LIN {X 42.103,Y -31.707,Z -45.890,A -90.000,B 90.000,C 0.000} C_DIS
LIN {X 42.764,Y -31.745,Z -45.727,A -90.000,B 90.000,C 0.000} C_DIS
LIN {X 43.314,Y -31.756,Z -45.575,A -90.000,B 90.000,C 0.000} C_DIS
LIN {X 43.681,Y -31.756,Z -45.477,A -90.000,B 90.000,C 0.000} C_DIS
LIN {X 44.130,Y -31.751,Z -45.363,A -90.000,B 90.000,C 0.000} C_DIS
LIN {X 44.222,Y -31.752,Z -45.341,A -90.000,B 90.000,C 0.000} C_DIS
LIN {X 44.913,Y -31.771,Z -45.188,A -90.000,B 90.000,C 0.000} C_DIS
LIN {X 45.364,Y -31.765,Z -45.111,A -90.000,B 90.000,C 0.000} C_DIS
LIN {X 45.432,Y -31.762,Z -45.099,A -90.000,B 90.000,C 0.000} C_DIS
LIN {X 45.844,Y -31.730,Z -45.045,A -90.000,B 90.000,C 0.000} C_DIS
LIN {X 45.937,Y -31.721,Z -45.037,A -90.000,B 90.000,C 0.000} C_DIS
LIN {X 46.177,Y -31.703,Z -45.019,A -90.000,B 90.000,C 0.000} C_DIS
LIN {X 46.589,Y -31.686,Z -44.979,A -90.000,B 90.000,C 0.000} C_DIS
LIN {X 46.721,Y -31.684,Z -44.970,A -90.000,B 90.000,C 0.000} C_DIS
LIN {X 47.117,Y -31.682,Z -44.943,A -90.000,B 90.000,C 0.000} C_DIS
LIN {X 47.760,Y -31.692,Z -44.913,A -90.000,B 90.000,C 0.000} C_DIS
LIN {X 48.195,Y -31.687,Z -44.927,A -90.000,B 90.000,C 0.000} C_DIS
LIN {X 48.804,Y -31.665,Z -44.973,A -90.000,B 90.000,C 0.000} C_DIS
LIN {X 49.258,Y -31.648,Z -45.032,A -90.000,B 90.000,C 0.000} C_DIS
LIN {X 49.697,Y -31.626,Z -45.108,A -90.000,B 90.000,C 0.000} C_DIS
LIN {X 49.817,Y -31.620,Z -45.134,A -90.000,B 90.000,C 0.000} C_DIS
LIN {X 50.403,Y -31.602,Z -45.264,A -90.000,B 90.000,C 0.000} C_DIS
LIN {X 50.513,Y -31.602,Z -45.290,A -90.000,B 90.000,C 0.000} C_DIS
LIN {X 50.923,Y -31.594,Z -45.415,A -90.000,B 90.000,C 0.000} C_DIS
LIN {X 51.695,Y -31.586,Z -45.677,A -90.000,B 90.000,C 0.000} C_DIS
LIN {X 52.507,Y -31.561,Z -46.005,A -90.000,B 90.000,C 0.000} C_DIS
LIN {X 52.949,Y -31.557,Z -46.198,A -90.000,B 90.000,C 0.000} C_DIS
LIN {X 53.402,Y -31.550,Z -46.401,A -90.000,B 90.000,C 0.000} C_DIS
LIN {X 53.812,Y -31.543,Z -46.594,A -90.000,B 90.000,C 0.000} C_DIS
LIN {X 54.024,Y -31.537,Z -46.700,A -90.000,B 90.000,C 0.000} C_DIS
LIN {X 54.190,Y -31.540,Z -46.786,A -90.000,B 90.000,C 0.000} C_DIS
LIN {X 54.466,Y -31.543,Z -46.938,A -90.000,B 90.000,C 0.000} C_DIS
LIN {X 54.513,Y -31.543,Z -46.967,A -90.000,B 90.000,C 0.000} C_DIS
LIN {X 54.861,Y -31.548,Z -47.185,A -90.000,B 90.000,C 0.000} C_DIS
LIN {X 55.840,Y -31.525,Z -47.889,A -90.000,B 90.000,C 0.000} C_DIS
LIN {X 57.235,Y -31.497,Z -48.888,A -90.000,B 90.000,C 0.000} C_DIS
LIN {X 57.411,Y -31.498,Z -49.016,A -90.000,B 90.000,C 0.000} C_DIS
LIN {X 57.592,Y -31.496,Z -49.156,A -90.000,B 90.000,C 0.000} C_DIS
LIN {X 57.780,Y -31.499,Z -49.303,A -90.000,B 90.000,C 0.000} C_DIS
LIN {X 59.169,Y -31.488,Z -50.515,A -90.000,B 90.000,C 0.000} C_DIS
LIN {X 60.060,Y -31.484,Z -51.286,A -90.000,B 90.000,C 0.000} C_DIS
LIN {X 60.371,Y -31.483,Z -51.578,A -90.000,B 90.000,C 0.000} C_DIS
LIN {X 61.487,Y -31.484,Z -52.631,A -90.000,B 90.000,C 0.000} C_DIS
LIN {X 62.016,Y -31.485,Z -53.126,A -90.000,B 90.000,C 0.000} C_DIS
LIN {X 62.615,Y -31.489,Z -53.684,A -90.000,B 90.000,C 0.000} C_DIS
LIN {X 63.420,Y -31.498,Z -54.433,A -90.000,B 90.000,C 0.000} C_DIS
LIN {X 64.379,Y -31.509,Z -55.331,A -90.000,B 90.000,C 0.000} C_DIS
LIN {X 64.718,Y -31.523,Z -55.625,A -90.000,B 90.000,C 0.000} C_DIS
LIN {X 65.056,Y -31.534,Z -55.917,A -90.000,B 90.000,C 0.000} C_DIS
LIN {X 65.997,Y -31.557,Z -56.726,A -90.000,B 90.000,C 0.000} C_DIS
LIN {X 66.900,Y -31.586,Z -57.486,A -90.000,B 90.000,C 0.000} C_DIS
LIN {X 67.393,Y -31.606,Z -57.902,A -90.000,B 90.000,C 0.000} C_DIS
LIN {X 68.612,Y -31.651,Z -58.950,A -90.000,B 90.000,C 0.000} C_DIS
LIN {X 69.045,Y -31.655,Z -59.347,A -90.000,B 90.000,C 0.000} C_DIS
LIN {X 69.869,Y -31.693,Z -60.129,A -90.000,B 90.000,C 0.000} C_DIS
LIN {X 70.229,Y -31.703,Z -60.488,A -90.000,B 90.000,C 0.000} C_DIS
LIN {X 70.602,Y -31.727,Z -60.873,A -90.000,B 90.000,C 0.000} C_DIS
LIN {X 71.184,Y -31.746,Z -61.521,A -90.000,B 90.000,C 0.000} C_DIS
LIN {X 72.241,Y -31.804,Z -62.721,A -90.000,B 90.000,C 0.000} C_DIS
LIN {X 72.515,Y -31.817,Z -63.037,A -90.000,B 90.000,C 0.000} C_DIS
LIN {X 72.609,Y -31.817,Z -63.151,A -90.000,B 90.000,C 0.000} C_DIS
LIN {X 72.801,Y -31.813,Z -63.398,A -90.000,B 90.000,C 0.000} C_DIS
LIN {X 72.929,Y -31.812,Z -63.565,A -90.000,B 90.000,C 0.000} C_DIS
LIN {X 73.104,Y -31.812,Z -63.793,A -90.000,B 90.000,C 0.000} C_DIS
LIN {X 73.529,Y -31.818,Z -64.361,A -90.000,B 90.000,C 0.000} C_DIS
LIN {X 73.683,Y -31.819,Z -64.579,A -90.000,B 90.000,C 0.000} C_DIS
LIN {X 73.927,Y -31.829,Z -64.916,A -90.000,B 90.000,C 0.000} C_DIS
LIN {X 73.994,Y -31.828,Z -65.015,A -90.000,B 90.000,C 0.000} C_DIS
LIN {X 74.219,Y -31.808,Z -65.329,A -90.000,B 90.000,C 0.000} C_DIS
LIN {X 74.431,Y -31.799,Z -65.639,A -90.000,B 90.000,C 0.000} C_DIS
LIN {X 74.577,Y -31.806,Z -65.839,A -90.000,B 90.000,C 0.000} C_DIS
LIN {X 74.823,Y -31.798,Z -66.153,A -90.000,B 90.000,C 0.000} C_DIS
LIN {X 74.927,Y -31.796,Z -66.289,A -90.000,B 90.000,C 0.000} C_DIS
LIN {X 75.187,Y -31.788,Z -66.638,A -90.000,B 90.000,C 0.000} C_DIS
LIN {X 75.305,Y -31.780,Z -66.797,A -90.000,B 90.000,C 0.000} C_DIS
LIN {X 75.814,Y -31.762,Z -67.510,A -90.000,B 90.000,C 0.000} C_DIS
LIN {X 75.836,Y -31.763,Z -67.538,A -90.000,B 90.000,C 0.000} C_DIS
LIN {X 75.961,Y -31.757,Z -67.682,A -90.000,B 90.000,C 0.000} C_DIS
LIN {X 76.227,Y -31.729,Z -68.017,A -90.000,B 90.000,C 0.000} C_DIS
LIN {X 76.293,Y -31.724,Z -68.107,A -90.000,B 90.000,C 0.000} C_DIS
LIN {X 76.429,Y -31.718,Z -68.299,A -90.000,B 90.000,C 0.000} C_DIS
LIN {X 76.455,Y -31.719,Z -68.332,A -90.000,B 90.000,C 0.000} C_DIS
LIN {X 76.904,Y -31.702,Z -68.861,A -90.000,B 90.000,C 0.000} C_DIS
LIN {X 76.997,Y -31.696,Z -68.977,A -90.000,B 90.000,C 0.000} C_DIS
LIN {X 77.105,Y -31.691,Z -69.109,A -90.000,B 90.000,C 0.000} C_DIS
LIN {X 77.203,Y -31.686,Z -69.228,A -90.000,B 90.000,C 0.000} C_DIS
LIN {X 77.430,Y -31.682,Z -69.512,A -90.000,B 90.000,C 0.000} C_DIS
LIN {X 77.622,Y -31.678,Z -69.759,A -90.000,B 90.000,C 0.000} C_DIS
LIN {X 77.717,Y -31.609,Z -69.804,A -90.000,B 90.000,C 0.000} C_DIS
LIN {X 77.780,Y -31.567,Z -69.838,A -90.000,B 90.000,C 0.000} C_DIS
LIN {X 77.852,Y -31.523,Z -69.884,A -90.000,B 90.000,C 0.000} C_DIS
LIN {X 77.939,Y -31.475,Z -69.946,A -90.000,B 90.000,C 0.000} C_DIS
LIN {X 78.032,Y -31.430,Z -70.019,A -90.000,B 90.000,C 0.000} C_DIS
LIN {X 78.096,Y -31.404,Z -70.072,A -90.000,B 90.000,C 0.000} C_DIS
LIN {X 78.244,Y -31.354,Z -70.211,A -90.000,B 90.000,C 0.000} C_DIS
LIN {X 78.265,Y -31.349,Z -70.232,A -90.000,B 90.000,C 0.000} C_DIS
LIN {X 78.399,Y -31.321,Z -70.376,A -90.000,B 90.000,C 0.000} C_DIS
LIN {X 78.478,Y -31.312,Z -70.466,A -90.000,B 90.000,C 0.000} C_DIS
LIN {X 78.570,Y -31.308,Z -70.580,A -90.000,B 90.000,C 0.000} C_DIS
LIN {X 78.560,Y -31.341,Z -70.590,A -90.000,B 90.000,C 0.000} C_DIS
LIN {X 78.561,Y -35.835,Z -70.592,A -90.000,B 90.000,C 0.000} C_DIS
LIN {X 78.567,Y -36.729,Z -70.599,A -90.000,B 90.000,C 0.000} C_DIS
LIN {X 78.574,Y -37.040,Z -70.607,A -90.000,B 90.000,C 0.000} C_DIS
LIN {X 78.584,Y -37.233,Z -70.617,A -90.000,B 90.000,C 0.000} C_DIS
LIN {X 78.578,Y -37.064,Z -70.596,A -90.000,B 90.000,C 0.000} C_DIS
LIN {X 78.575,Y -36.863,Z -70.579,A -90.000,B 90.000,C 0.000} C_DIS
LIN {X 78.573,Y -35.838,Z -70.554,A -90.000,B 90.000,C 0.000} C_DIS
LIN {X 78.573,Y -31.307,Z -70.553,A -90.000,B 90.000,C 0.000} C_DIS
LIN {X 78.577,Y -31.307,Z -70.516,A -90.000,B 90.000,C 0.000} C_DIS
LIN {X 78.594,Y -31.308,Z -70.505,A -90.000,B 90.000,C 0.000} C_DIS
LIN {X 78.624,Y -31.308,Z -70.415,A -90.000,B 90.000,C 0.000} C_DIS
LIN {X 78.683,Y -36.449,Z -70.235,A -90.000,B 90.000,C 0.000} C_DIS
LIN {X 78.690,Y -36.457,Z -70.213,A -90.000,B 90.000,C 0.000} C_DIS
LIN {X 78.691,Y -36.460,Z -70.211,A -90.000,B 90.000,C 0.000} C_DIS
LIN {X 78.693,Y -36.503,Z -70.206,A -90.000,B 90.000,C 0.000} C_DIS
LIN {X 78.701,Y -36.545,Z -70.184,A -90.000,B 90.000,C 0.000} C_DIS
LIN {X 78.761,Y -31.308,Z -70.004,A -90.000,B 90.000,C 0.000} C_DIS
LIN {X 78.774,Y -31.308,Z -69.967,A -90.000,B 90.000,C 0.000} C_DIS
LIN {X 78.774,Y -60.000,Z -69.967,A -90.000,B 90.000,C 0.000} C_DIS
LIN {X 87.886,Y -60.000,Z -55.601,A -90.000,B 90.000,C 0.000} C_DIS
LIN {X 87.886,Y -31.308,Z -55.601,A -90.000,B 90.000,C 0.000} C_DIS
LIN {X 87.895,Y -31.310,Z -55.489,A -90.000,B 90.000,C 0.000} C_DIS
LIN {X 87.955,Y -31.321,Z -55.235,A -90.000,B 90.000,C 0.000} C_DIS
LIN {X 88.019,Y -31.333,Z -55.056,A -90.000,B 90.000,C 0.000} C_DIS
LIN {X 88.137,Y -31.354,Z -54.797,A -90.000,B 90.000,C 0.000} C_DIS
LIN {X 88.416,Y -31.405,Z -54.284,A -90.000,B 90.000,C 0.000} C_DIS
LIN {X 88.556,Y -31.441,Z -54.017,A -90.000,B 90.000,C 0.000} C_DIS
LIN {X 88.594,Y -31.451,Z -53.947,A -90.000,B 90.000,C 0.000} C_DIS
LIN {X 88.969,Y -31.547,Z -53.327,A -90.000,B 90.000,C 0.000} C_DIS
LIN {X 89.043,Y -31.566,Z -53.212,A -90.000,B 90.000,C 0.000} C_DIS
LIN {X 89.236,Y -31.615,Z -52.925,A -90.000,B 90.000,C 0.000} C_DIS
LIN {X 89.391,Y -31.655,Z -52.704,A -90.000,B 90.000,C 0.000} C_DIS
LIN {X 89.464,Y -31.674,Z -52.605,A -90.000,B 90.000,C 0.000} C_DIS
LIN {X 89.839,Y -31.793,Z -52.083,A -90.000,B 90.000,C 0.000} C_DIS
LIN {X 90.193,Y -31.904,Z -51.622,A -90.000,B 90.000,C 0.000} C_DIS
LIN {X 90.500,Y -32.000,Z -51.242,A -90.000,B 90.000,C 0.000} C_DIS
LIN {X 90.638,Y -32.043,Z -51.076,A -90.000,B 90.000,C 0.000} C_DIS
LIN {X 91.176,Y -32.230,Z -50.436,A -90.000,B 90.000,C 0.000} C_DIS
LIN {X 91.462,Y -32.330,Z -50.116,A -90.000,B 90.000,C 0.000} C_DIS
LIN {X 91.851,Y -32.466,Z -49.697,A -90.000,B 90.000,C 0.000} C_DIS
LIN {X 92.169,Y -32.589,Z -49.359,A -90.000,B 90.000,C 0.000} C_DIS
LIN {X 92.399,Y -32.678,Z -49.123,A -90.000,B 90.000,C 0.000} C_DIS
LIN {X 92.339,Y -32.668,Z -48.928,A -90.000,B 90.000,C 0.000} C_DIS
LIN {X 92.298,Y -32.662,Z -48.770,A -90.000,B 90.000,C 0.000} C_DIS
LIN {X 92.252,Y -32.641,Z -48.535,A -90.000,B 90.000,C 0.000} C_DIS
LIN {X 92.218,Y -32.617,Z -48.349,A -90.000,B 90.000,C 0.000} C_DIS
LIN {X 92.177,Y -32.587,Z -48.082,A -90.000,B 90.000,C 0.000} C_DIS
LIN {X 92.166,Y -32.569,Z -47.976,A -90.000,B 90.000,C 0.000} C_DIS
LIN {X 92.158,Y -32.552,Z -47.869,A -90.000,B 90.000,C 0.000} C_DIS
LIN {X 92.148,Y -32.512,Z -47.664,A -90.000,B 90.000,C 0.000} C_DIS
LIN {X 92.146,Y -32.500,Z -47.597,A -90.000,B 90.000,C 0.000} C_DIS
LIN {X 92.150,Y -32.478,Z -47.451,A -90.000,B 90.000,C 0.000} C_DIS
LIN {X 92.171,Y -32.438,Z -47.211,A -90.000,B 90.000,C 0.000} C_DIS
LIN {X 92.200,Y -32.388,Z -46.981,A -90.000,B 90.000,C 0.000} C_DIS
LIN {X 92.221,Y -32.361,Z -46.845,A -90.000,B 90.000,C 0.000} C_DIS
LIN {X 92.284,Y -32.302,Z -46.521,A -90.000,B 90.000,C 0.000} C_DIS
LIN {X 92.307,Y -32.284,Z -46.424,A -90.000,B 90.000,C 0.000} C_DIS
LIN {X 92.324,Y -32.273,Z -46.362,A -90.000,B 90.000,C 0.000} C_DIS
LIN {X 92.409,Y -32.240,Z -46.102,A -90.000,B 90.000,C 0.000} C_DIS
LIN {X 92.452,Y -32.221,Z -45.979,A -90.000,B 90.000,C 0.000} C_DIS
LIN {X 92.675,Y -32.135,Z -45.409,A -90.000,B 90.000,C 0.000} C_DIS
LIN {X 92.727,Y -32.118,Z -45.300,A -90.000,B 90.000,C 0.000} C_DIS
LIN {X 92.805,Y -32.095,Z -45.145,A -90.000,B 90.000,C 0.000} C_DIS
LIN {X 92.914,Y -32.062,Z -44.937,A -90.000,B 90.000,C 0.000} C_DIS
LIN {X 93.148,Y -32.006,Z -44.518,A -90.000,B 90.000,C 0.000} C_DIS
LIN {X 93.166,Y -32.002,Z -44.486,A -90.000,B 90.000,C 0.000} C_DIS
LIN {X 93.389,Y -31.943,Z -44.141,A -90.000,B 90.000,C 0.000} C_DIS
LIN {X 93.591,Y -31.898,Z -43.848,A -90.000,B 90.000,C 0.000} C_DIS
LIN {X 93.761,Y -31.866,Z -43.610,A -90.000,B 90.000,C 0.000} C_DIS
LIN {X 94.205,Y -31.773,Z -43.062,A -90.000,B 90.000,C 0.000} C_DIS
LIN {X 94.307,Y -31.752,Z -42.942,A -90.000,B 90.000,C 0.000} C_DIS
LIN {X 94.451,Y -31.729,Z -42.780,A -90.000,B 90.000,C 0.000} C_DIS
LIN {X 94.667,Y -31.693,Z -42.552,A -90.000,B 90.000,C 0.000} C_DIS
LIN {X 94.923,Y -31.657,Z -42.285,A -90.000,B 90.000,C 0.000} C_DIS
LIN {X 95.182,Y -31.617,Z -42.030,A -90.000,B 90.000,C 0.000} C_DIS
LIN {X 95.304,Y -31.603,Z -41.920,A -90.000,B 90.000,C 0.000} C_DIS
LIN {X 95.776,Y -31.549,Z -41.516,A -90.000,B 90.000,C 0.000} C_DIS
LIN {X 95.980,Y -31.527,Z -41.343,A -90.000,B 90.000,C 0.000} C_DIS
LIN {X 96.207,Y -31.500,Z -41.168,A -90.000,B 90.000,C 0.000} C_DIS
LIN {X 96.826,Y -31.455,Z -40.703,A -90.000,B 90.000,C 0.000} C_DIS
LIN {X 96.924,Y -31.447,Z -40.637,A -90.000,B 90.000,C 0.000} C_DIS
LIN {X 97.187,Y -31.423,Z -40.470,A -90.000,B 90.000,C 0.000} C_DIS
LIN {X 97.655,Y -31.396,Z -40.178,A -90.000,B 90.000,C 0.000} C_DIS
LIN {X 98.035,Y -31.375,Z -39.949,A -90.000,B 90.000,C 0.000} C_DIS
LIN {X 98.217,Y -31.365,Z -39.850,A -90.000,B 90.000,C 0.000} C_DIS
LIN {X 98.843,Y -31.345,Z -39.508,A -90.000,B 90.000,C 0.000} C_DIS
LIN {X 99.070,Y -31.336,Z -39.398,A -90.000,B 90.000,C 0.000} C_DIS
LIN {X 99.520,Y -31.325,Z -39.184,A -90.000,B 90.000,C 0.000} C_DIS
LIN {X 100.000,Y -31.317,Z -38.956,A -90.000,B 90.000,C 0.000} C_DIS
LIN {X 100.283,Y -31.314,Z -38.822,A -90.000,B 90.000,C 0.000} C_DIS
LIN {X 101.144,Y -31.310,Z -38.432,A -90.000,B 90.000,C 0.000} C_DIS
LIN {X 102.050,Y -31.308,Z -38.021,A -90.000,B 90.000,C 0.000} C_DIS
LIN {X 102.908,Y -31.316,Z -37.638,A -90.000,B 90.000,C 0.000} C_DIS
LIN {X 103.020,Y -31.308,Z -37.588,A -90.000,B 90.000,C 0.000} C_DIS
LIN {X 103.177,Y -31.308,Z -37.517,A -90.000,B 90.000,C 0.000} C_DIS
LIN {X 103.228,Y -31.308,Z -37.495,A -90.000,B 90.000,C 0.000} C_DIS
LIN {X 103.228,Y -60.000,Z -37.495,A -90.000,B 90.000,C 0.000} C_DIS
LIN {X 117.072,Y -60.000,Z -39.281,A -90.000,B 90.000,C 0.000} C_DIS
LIN {X 117.072,Y -31.308,Z -39.281,A -90.000,B 90.000,C 0.000} C_DIS
LIN {X 117.089,Y -31.308,Z -39.324,A -90.000,B 90.000,C 0.000} C_DIS
LIN {X 117.313,Y -31.308,Z -39.869,A -90.000,B 90.000,C 0.000} C_DIS
LIN {X 117.419,Y -31.307,Z -40.116,A -90.000,B 90.000,C 0.000} C_DIS
LIN {X 117.617,Y -31.305,Z -40.562,A -90.000,B 90.000,C 0.000} C_DIS
LIN {X 117.799,Y -31.303,Z -40.949,A -90.000,B 90.000,C 0.000} C_DIS
LIN {X 117.883,Y -31.301,Z -41.121,A -90.000,B 90.000,C 0.000} C_DIS
LIN {X 118.041,Y -31.298,Z -41.427,A -90.000,B 90.000,C 0.000} C_DIS
LIN {X 118.113,Y -31.296,Z -41.562,A -90.000,B 90.000,C 0.000} C_DIS
LIN {X 118.247,Y -31.291,Z -41.796,A -90.000,B 90.000,C 0.000} C_DIS
LIN {X 118.418,Y -31.284,Z -42.072,A -90.000,B 90.000,C 0.000} C_DIS
LIN {X 118.513,Y -31.279,Z -42.211,A -90.000,B 90.000,C 0.000} C_DIS
LIN {X 118.593,Y -31.273,Z -42.319,A -90.000,B 90.000,C 0.000} C_DIS
LIN {X 118.659,Y -31.268,Z -42.401,A -90.000,B 90.000,C 0.000} C_DIS
LIN {X 118.761,Y -31.255,Z -42.521,A -90.000,B 90.000,C 0.000} C_DIS
LIN {X 118.778,Y -31.250,Z -42.546,A -90.000,B 90.000,C 0.000} C_DIS
LIN {X 118.782,Y -31.245,Z -42.566,A -90.000,B 90.000,C 0.000} C_DIS
LIN {X 118.779,Y -31.243,Z -42.575,A -90.000,B 90.000,C 0.000} C_DIS
LIN {X 118.764,Y -31.239,Z -42.594,A -90.000,B 90.000,C 0.000} C_DIS
LIN {X 118.671,Y -31.233,Z -42.672,A -90.000,B 90.000,C 0.000} C_DIS
LIN {X 118.579,Y -31.231,Z -42.764,A -90.000,B 90.000,C 0.000} C_DIS
LIN {X 118.504,Y -31.231,Z -42.852,A -90.000,B 90.000,C 0.000} C_DIS
LIN {X 118.418,Y -31.233,Z -42.968,A -90.000,B 90.000,C 0.000} C_DIS
LIN {X 118.321,Y -31.235,Z -43.116,A -90.000,B 90.000,C 0.000} C_DIS
LIN {X 118.213,Y -31.239,Z -43.300,A -90.000,B 90.000,C 0.000} C_DIS
LIN {X 118.095,Y -31.244,Z -43.525,A -90.000,B 90.000,C 0.000} C_DIS
LIN {X 118.033,Y -31.247,Z -43.654,A -90.000,B 90.000,C 0.000} C_DIS
LIN {X 117.900,Y -31.254,Z -43.948,A -90.000,B 90.000,C 0.000} C_DIS
LIN {X 117.830,Y -31.259,Z -44.114,A -90.000,B 90.000,C 0.000} C_DIS
LIN {X 117.683,Y -31.268,Z -44.488,A -90.000,B 90.000,C 0.000} C_DIS
LIN {X 117.606,Y -31.274,Z -44.696,A -90.000,B 90.000,C 0.000} C_DIS
LIN {X 117.446,Y -31.286,Z -45.159,A -90.000,B 90.000,C 0.000} C_DIS
LIN {X 117.363,Y -31.293,Z -45.415,A -90.000,B 90.000,C 0.000} C_DIS
LIN {X 117.189,Y -31.308,Z -45.978,A -90.000,B 90.000,C 0.000} C_DIS
LIN {X 117.160,Y -31.311,Z -46.076,A -90.000,B 90.000,C 0.000} C_DIS
LIN {X 117.121,Y -31.308,Z -46.207,A -90.000,B 90.000,C 0.000} C_DIS
LIN {X 117.121,Y -60.000,Z -46.207,A -90.000,B 90.000,C 0.000} C_DIS
LIN {X 112.812,Y -60.000,Z -55.800,A -90.000,B 90.000,C 0.000} C_DIS
LIN {X 112.812,Y -31.308,Z -55.800,A -90.000,B 90.000,C 0.000} C_DIS
LIN {X 112.799,Y -31.308,Z -55.830,A -90.000,B 90.000,C 0.000} C_DIS
LIN {X 112.799,Y -60.000,Z -55.830,A -90.000,B 90.000,C 0.000} C_DIS
LIN {X 88.972,Y -60.000,Z -50.129,A -90.000,B 90.000,C 0.000} C_DIS
LIN {X 88.972,Y -31.308,Z -50.129,A -90.000,B 90.000,C 0.000} C_DIS
LIN {X 89.131,Y -31.353,Z -49.936,A -90.000,B 90.000,C 0.000} C_DIS
LIN {X 89.286,Y -31.397,Z -49.752,A -90.000,B 90.000,C 0.000} C_DIS
LIN {X 89.455,Y -31.446,Z -49.556,A -90.000,B 90.000,C 0.000} C_DIS
LIN {X 89.833,Y -31.552,Z -49.118,A -90.000,B 90.000,C 0.000} C_DIS
LIN {X 90.193,Y -31.659,Z -48.723,A -90.000,B 90.000,C 0.000} C_DIS
LIN {X 90.416,Y -31.728,Z -48.487,A -90.000,B 90.000,C 0.000} C_DIS
LIN {X 90.410,Y -31.670,Z -48.304,A -90.000,B 90.000,C 0.000} C_DIS
LIN {X 90.409,Y -31.620,Z -48.138,A -90.000,B 90.000,C 0.000} C_DIS
LIN {X 90.414,Y -31.537,Z -47.877,A -90.000,B 90.000,C 0.000} C_DIS
LIN {X 90.420,Y -31.503,Z -47.762,A -90.000,B 90.000,C 0.000} C_DIS
LIN {X 90.432,Y -31.468,Z -47.635,A -90.000,B 90.000,C 0.000} C_DIS
LIN {X 90.455,Y -31.417,Z -47.473,A -90.000,B 90.000,C 0.000} C_DIS
LIN {X 90.518,Y -31.308,Z -47.110,A -90.000,B 90.000,C 0.000} C_DIS
LIN {X 90.518,Y -60.000,Z -47.110,A -90.000,B 90.000,C 0.000} C_DIS
LIN {X -51.676,Y -60.000,Z -94.928,A -90.000,B 90.000,C 0.000} C_DIS
LIN {X -51.676,Y -31.308,Z -94.928,A -90.000,B 90.000,C 0.000} C_DIS
LIN {X -52.105,Y -31.387,Z -94.074,A -90.000,B 90.000,C 0.000} C_DIS
LIN {X -52.393,Y -31.436,Z -93.493,A -90.000,B 90.000,C 0.000} C_DIS
LIN {X -52.925,Y -31.509,Z -92.389,A -90.000,B 90.000,C 0.000} C_DIS
LIN {X -53.030,Y -31.517,Z -92.158,A -90.000,B 90.000,C 0.000} C_DIS
LIN {X -53.230,Y -31.540,Z -91.682,A -90.000,B 90.000,C 0.000} C_DIS
LIN {X -53.482,Y -31.581,Z -91.035,A -90.000,B 90.000,C 0.000} C_DIS
LIN {X -53.607,Y -31.607,Z -90.689,A -90.000,B 90.000,C 0.000} C_DIS
LIN {X -54.074,Y -31.717,Z -89.348,A -90.000,B 90.000,C 0.000} C_DIS
LIN {X -54.336,Y -31.775,Z -88.604,A -90.000,B 90.000,C 0.000} C_DIS
LIN {X -54.457,Y -31.803,Z -88.253,A -90.000,B 90.000,C 0.000} C_DIS
LIN {X -54.652,Y -31.821,Z -87.641,A -90.000,B 90.000,C 0.000} C_DIS
LIN {X -54.746,Y -31.832,Z -87.327,A -90.000,B 90.000,C 0.000} C_DIS
LIN {X -54.932,Y -31.854,Z -86.694,A -90.000,B 90.000,C 0.000} C_DIS
LIN {X -55.381,Y -31.918,Z -85.161,A -90.000,B 90.000,C 0.000} C_DIS
LIN {X -55.413,Y -31.924,Z -85.040,A -90.000,B 90.000,C 0.000} C_DIS
LIN {X -55.466,Y -31.938,Z -84.818,A -90.000,B 90.000,C 0.000} C_DIS
LIN {X -55.521,Y -31.946,Z -84.578,A -90.000,B 90.000,C 0.000} C_DIS
LIN {X -55.916,Y -31.978,Z -82.819,A -90.000,B 90.000,C 0.000} C_DIS
LIN {X -56.007,Y -31.991,Z -82.356,A -90.000,B 90.000,C 0.000} C_DIS
LIN {X -56.250,Y -32.045,Z -81.134,A -90.000,B 90.000,C 0.000} C_DIS
LIN {X -56.270,Y -32.049,Z -81.032,A -90.000,B 90.000,C 0.000} C_DIS
LIN {X -56.329,Y -32.059,Z -80.716,A -90.000,B 90.000,C 0.000} C_DIS
LIN {X -56.379,Y -32.073,Z -80.395,A -90.000,B 90.000,C 0.000} C_DIS
LIN {X -56.448,Y -32.106,Z -79.815,A -90.000,B 90.000,C 0.000} C_DIS
LIN {X -56.504,Y -32.125,Z -79.294,A -90.000,B 90.000,C 0.000} C_DIS
LIN {X -56.603,Y -32.155,Z -78.446,A -90.000,B 90.000,C 0.000} C_DIS
LIN {X -56.621,Y -32.163,Z -78.205,A -90.000,B 90.000,C 0.000} C_DIS
LIN {X -56.659,Y -32.219,Z -77.292,A -90.000,B 90.000,C 0.000} C_DIS
LIN {X -56.673,Y -32.236,Z -76.915,A -90.000,B 90.000,C 0.000} C_DIS
LIN {X -56.683,Y -32.255,Z -76.513,A -90.000,B 90.000,C 0.000} C_DIS
LIN {X -56.684,Y -32.260,Z -76.417,A -90.000,B 90.000,C 0.000} C_DIS
LIN {X -56.698,Y -32.266,Z -76.248,A -90.000,B 90.000,C 0.000} C_DIS
LIN {X -56.702,Y -32.271,Z -76.134,A -90.000,B 90.000,C 0.000} C_DIS
LIN {X -56.708,Y -32.294,Z -75.585,A -90.000,B 90.000,C 0.000} C_DIS
LIN {X -56.715,Y -32.320,Z -74.894,A -90.000,B 90.000,C 0.000} C_DIS
LIN {X -56.730,Y -32.326,Z -74.671,A -90.000,B 90.000,C 0.000} C_DIS
LIN {X -56.736,Y -32.331,Z -74.526,A -90.000,B 90.000,C 0.000} C_DIS
LIN {X -56.737,Y -32.336,Z -74.426,A -90.000,B 90.000,C 0.000} C_DIS
LIN {X -56.729,Y -32.346,Z -74.196,A -90.000,B 90.000,C 0.000} C_DIS
LIN {X -56.692,Y -32.368,Z -73.660,A -90.000,B 90.000,C 0.000} C_DIS
LIN {X -56.665,Y -32.392,Z -73.248,A -90.000,B 90.000,C 0.000} C_DIS
LIN {X -56.672,Y -32.402,Z -72.968,A -90.000,B 90.000,C 0.000} C_DIS
LIN {X -56.670,Y -32.409,Z -72.764,A -90.000,B 90.000,C 0.000} C_DIS
LIN {X -56.638,Y -32.420,Z -72.335,A -90.000,B 90.000,C 0.000} C_DIS
LIN {X -56.613,Y -32.433,Z -72.116,A -90.000,B 90.000,C 0.000} C_DIS
LIN {X -56.519,Y -32.475,Z -71.506,A -90.000,B 90.000,C 0.000} C_DIS
LIN {X -56.500,Y -32.479,Z -71.389,A -90.000,B 90.000,C 0.000} C_DIS
LIN {X -56.487,Y -32.481,Z -71.149,A -90.000,B 90.000,C 0.000} C_DIS
LIN {X -56.476,Y -32.482,Z -71.025,A -90.000,B 90.000,C 0.000} C_DIS
LIN {X -56.462,Y -32.490,Z -70.849,A -90.000,B 90.000,C 0.000} C_DIS
LIN {X -56.413,Y -32.508,Z -70.510,A -90.000,B 90.000,C 0.000} C_DIS
LIN {X -56.388,Y -32.517,Z -70.373,A -90.000,B 90.000,C 0.000} C_DIS
LIN {X -56.339,Y -32.531,Z -70.175,A -90.000,B 90.000,C 0.000} C_DIS
LIN {X -56.286,Y -32.540,Z -69.977,A -90.000,B 90.000,C 0.000} C_DIS
LIN {X -56.232,Y -32.546,Z -69.782,A -90.000,B 90.000,C 0.000} C_DIS
LIN {X -56.174,Y -32.559,Z -69.566,A -90.000,B 90.000,C 0.000} C_DIS
LIN {X -56.125,Y -32.572,Z -69.221,A -90.000,B 90.000,C 0.000} C_DIS
LIN {X -56.095,Y -32.579,Z -69.061,A -90.000,B 90.000,C 0.000} C_DIS
LIN {X -56.029,Y -32.593,Z -68.796,A -90.000,B 90.000,C 0.000} C_DIS
LIN {X -55.977,Y -32.595,Z -68.621,A -90.000,B 90.000,C 0.000} C_DIS
LIN {X -55.932,Y -32.594,Z -68.474,A -90.000,B 90.000,C 0.000} C_DIS
LIN {X -55.877,Y -32.598,Z -68.325,A -90.000,B 90.000,C 0.000} C_DIS
LIN {X -55.745,Y -32.611,Z -67.997,A -90.000,B 90.000,C 0.000} C_DIS
LIN {X -55.685,Y -32.617,Z -67.868,A -90.000,B 90.000,C 0.000} C_DIS
LIN {X -55.515,Y -32.634,Z -67.534,A -90.000,B 90.000,C 0.000} C_DIS
LIN {X -55.433,Y -32.633,Z -67.375,A -90.000,B 90.000,C 0.000} C_DIS
LIN {X -55.378,Y -32.628,Z -67.269,A -90.000,B 90.000,C 0.000} C_DIS
LIN {X -55.298,Y -32.615,Z -67.062,A -90.000,B 90.000,C 0.000} C_DIS
LIN {X -55.209,Y -32.609,Z -66.858,A -90.000,B 90.000,C 0.000} C_DIS
LIN {X -55.129,Y -32.605,Z -66.697,A -90.000,B 90.000,C 0.000} C_DIS
LIN {X -54.902,Y -32.599,Z -66.282,A -90.000,B 90.000,C 0.000} C_DIS
LIN {X -54.820,Y -32.593,Z -66.148,A -90.000,B 90.000,C 0.000} C_DIS
LIN {X -54.729,Y -32.582,Z -66.010,A -90.000,B 90.000,C 0.000} C_DIS
LIN {X -54.612,Y -32.571,Z -65.851,A -90.000,B 90.000,C 0.000} C_DIS
LIN {X -54.560,Y -32.567,Z -65.785,A -90.000,B 90.000,C 0.000} C_DIS
LIN {X -54.405,Y -32.548,Z -65.605,A -90.000,B 90.000,C 0.000} C_DIS
LIN {X -54.268,Y -32.533,Z -65.452,A -90.000,B 90.000,C 0.000} C_DIS
LIN {X -54.208,Y -32.527,Z -65.388,A -90.000,B 90.000,C 0.000} C_DIS
LIN {X -53.880,Y -32.498,Z -65.053,A -90.000,B 90.000,C 0.000} C_DIS
LIN {X -53.575,Y -32.477,Z -64.741,A -90.000,B 90.000,C 0.000} C_DIS
LIN {X -53.460,Y -32.464,Z -64.626,A -90.000,B 90.000,C 0.000} C_DIS
LIN {X -53.029,Y -32.377,Z -64.202,A -90.000,B 90.000,C 0.000} C_DIS
LIN {X -52.891,Y -32.352,Z -64.077,A -90.000,B 90.000,C 0.000} C_DIS
LIN {X -52.829,Y -32.342,Z -64.025,A -90.000,B 90.000,C 0.000} C_DIS
LIN {X -52.651,Y -32.316,Z -63.884,A -90.000,B 90.000,C 0.000} C_DIS
LIN {X -52.325,Y -32.278,Z -63.652,A -90.000,B 90.000,C 0.000} C_DIS
LIN {X -52.210,Y -32.267,Z -63.576,A -90.000,B 90.000,C 0.000} C_DIS
LIN {X -52.068,Y -32.254,Z -63.487,A -90.000,B 90.000,C 0.000} C_DIS
LIN {X -51.593,Y -32.205,Z -63.173,A -90.000,B 90.000,C 0.000} C_DIS
LIN {X -51.197,Y -32.143,Z -62.921,A -90.000,B 90.000,C 0.000} C_DIS
LIN {X -51.009,Y -32.116,Z -62.808,A -90.000,B 90.000,C 0.000} C_DIS
LIN {X -50.538,Y -32.056,Z -62.543,A -90.000,B 90.000,C 0.000} C_DIS
LIN {X -50.324,Y -32.032,Z -62.429,A -90.000,B 90.000,C 0.000} C_DIS
LIN {X -49.822,Y -31.985,Z -62.188,A -90.000,B 90.000,C 0.000} C_DIS
LIN {X -49.461,Y -31.943,Z -62.023,A -90.000,B 90.000,C 0.000} C_DIS
LIN {X -49.322,Y -31.929,Z -61.967,A -90.000,B 90.000,C 0.000} C_DIS
LIN {X -49.113,Y -31.913,Z -61.890,A -90.000,B 90.000,C 0.000} C_DIS
LIN {X -47.888,Y -31.840,Z -61.477,A -90.000,B 90.000,C 0.000} C_DIS
LIN {X -46.739,Y -31.766,Z -61.084,A -90.000,B 90.000,C 0.000} C_DIS
LIN {X -46.546,Y -31.755,Z -61.022,A -90.000,B 90.000,C 0.000} C_DIS
LIN {X -46.153,Y -31.737,Z -60.912,A -90.000,B 90.000,C 0.000} C_DIS
LIN {X -45.452,Y -31.702,Z -60.734,A -90.000,B 90.000,C 0.000} C_DIS
LIN {X -44.255,Y -31.658,Z -60.469,A -90.000,B 90.000,C 0.000} C_DIS
LIN {X -43.968,Y -31.652,Z -60.405,A -90.000,B 90.000,C 0.000} C_DIS
LIN {X -43.761,Y -31.644,Z -60.363,A -90.000,B 90.000,C 0.000} C_DIS
LIN {X -41.648,Y -31.567,Z -59.998,A -90.000,B 90.000,C 0.000} C_DIS
LIN {X -41.394,Y -31.556,Z -59.957,A -90.000,B 90.000,C 0.000} C_DIS
LIN {X -41.350,Y -31.555,Z -59.952,A -90.000,B 90.000,C 0.000} C_DIS
LIN {X -40.374,Y -31.480,Z -59.871,A -90.000,B 90.000,C 0.000} C_DIS
LIN {X -40.133,Y -31.467,Z -59.858,A -90.000,B 90.000,C 0.000} C_DIS
LIN {X -39.781,Y -31.453,Z -59.843,A -90.000,B 90.000,C 0.000} C_DIS
LIN {X -39.621,Y -31.448,Z -59.841,A -90.000,B 90.000,C 0.000} C_DIS
LIN {X -39.390,Y -31.441,Z -59.838,A -90.000,B 90.000,C 0.000} C_DIS
LIN {X -38.631,Y -31.405,Z -59.821,A -90.000,B 90.000,C 0.000} C_DIS
LIN {X -38.474,Y -31.396,Z -59.818,A -90.000,B 90.000,C 0.000} C_DIS
LIN {X -37.801,Y -31.323,Z -59.826,A -90.000,B 90.000,C 0.000} C_DIS
LIN {X -37.674,Y -31.308,Z -59.829,A -90.000,B 90.000,C 0.000} C_DIS
LIN {X -37.674,Y -60.000,Z -59.829,A -90.000,B 90.000,C 0.000} C_DIS
LIN {X -57.638,Y -60.000,Z -83.771,A -90.000,B 90.000,C 0.000} C_DIS
LIN {X -57.638,Y -31.308,Z -83.771,A -90.000,B 90.000,C 0.000} C_DIS
LIN {X -57.786,Y -31.358,Z -83.168,A -90.000,B 90.000,C 0.000} C_DIS
LIN {X -57.882,Y -31.400,Z -82.724,A -90.000,B 90.000,C 0.000} C_DIS
LIN {X -58.063,Y -31.442,Z -81.818,A -90.000,B 90.000,C 0.000} C_DIS
LIN {X -58.212,Y -31.475,Z -81.053,A -90.000,B 90.000,C 0.000} C_DIS
LIN {X -58.268,Y -31.495,Z -80.707,A -90.000,B 90.000,C 0.000} C_DIS
LIN {X -58.287,Y -31.504,Z -80.584,A -90.000,B 90.000,C 0.000} C_DIS
LIN {X -58.318,Y -31.524,Z -80.340,A -90.000,B 90.000,C 0.000} C_DIS
LIN {X -58.432,Y -31.593,Z -79.391,A -90.000,B 90.000,C 0.000} C_DIS
LIN {X -58.527,Y -31.640,Z -78.631,A -90.000,B 90.000,C 0.000} C_DIS
LIN {X -58.552,Y -31.659,Z -78.334,A -90.000,B 90.000,C 0.000} C_DIS
LIN {X -58.566,Y -31.679,Z -78.071,A -90.000,B 90.000,C 0.000} C_DIS
LIN {X -58.611,Y -31.747,Z -76.979,A -90.000,B 90.000,C 0.000} C_DIS
LIN {X -58.623,Y -31.771,Z -76.489,A -90.000,B 90.000,C 0.000} C_DIS
LIN {X -58.632,Y -31.775,Z -76.385,A -90.000,B 90.000,C 0.000} C_DIS
LIN {X -58.643,Y -31.786,Z -76.135,A -90.000,B 90.000,C 0.000} C_DIS
LIN {X -58.651,Y -31.820,Z -75.471,A -90.000,B 90.000,C 0.000} C_DIS
LIN {X -58.658,Y -31.848,Z -74.959,A -90.000,B 90.000,C 0.000} C_DIS
LIN {X -58.665,Y -31.852,Z -74.858,A -90.000,B 90.000,C 0.000} C_DIS
LIN {X -58.674,Y -31.858,Z -74.720,A -90.000,B 90.000,C 0.000} C_DIS
LIN {X -58.682,Y -31.868,Z -74.485,A -90.000,B 90.000,C 0.000} C_DIS
LIN {X -58.681,Y -31.878,Z -74.303,A -90.000,B 90.000,C 0.000} C_DIS
LIN {X -58.671,Y -31.894,Z -74.044,A -90.000,B 90.000,C 0.000} C_DIS
LIN {X -58.641,Y -31.928,Z -73.559,A -90.000,B 90.000,C 0.000} C_DIS
LIN {X -58.617,Y -31.953,Z -73.188,A -90.000,B 90.000,C 0.000} C_DIS
LIN {X -58.623,Y -31.964,Z -72.932,A -90.000,B 90.000,C 0.000} C_DIS
LIN {X -58.621,Y -31.974,Z -72.728,A -90.000,B 90.000,C 0.000} C_DIS
LIN {X -58.616,Y -31.982,Z -72.588,A -90.000,B 90.000,C 0.000} C_DIS
LIN {X -58.592,Y -32.012,Z -72.212,A -90.000,B 90.000,C 0.000} C_DIS
LIN {X -58.583,Y -32.018,Z -72.095,A -90.000,B 90.000,C 0.000} C_DIS
LIN {X -58.547,Y -32.038,Z -71.791,A -90.000,B 90.000,C 0.000} C_DIS
LIN {X -58.490,Y -32.064,Z -71.424,A -90.000,B 90.000,C 0.000} C_DIS
LIN {X -58.452,Y -32.089,Z -71.168,A -90.000,B 90.000,C 0.000} C_DIS
LIN {X -58.446,Y -32.100,Z -71.021,A -90.000,B 90.000,C 0.000} C_DIS
LIN {X -58.419,Y -32.115,Z -70.675,A -90.000,B 90.000,C 0.000} C_DIS
LIN {X -58.405,Y -32.122,Z -70.548,A -90.000,B 90.000,C 0.000} C_DIS
LIN {X -58.360,Y -32.140,Z -70.236,A -90.000,B 90.000,C 0.000} C_DIS
LIN {X -58.336,Y -32.154,Z -70.089,A -90.000,B 90.000,C 0.000} C_DIS
LIN {X -58.297,Y -32.174,Z -69.887,A -90.000,B 90.000,C 0.000} C_DIS
LIN {X -58.226,Y -32.203,Z -69.598,A -90.000,B 90.000,C 0.000} C_DIS
LIN {X -58.107,Y -32.229,Z -69.155,A -90.000,B 90.000,C 0.000} C_DIS
LIN {X -58.093,Y -32.233,Z -69.054,A -90.000,B 90.000,C 0.000} C_DIS
LIN {X -58.062,Y -32.250,Z -68.841,A -90.000,B 90.000,C 0.000} C_DIS
LIN {X -58.028,Y -32.266,Z -68.653,A -90.000,B 90.000,C 0.000} C_DIS
LIN {X -57.992,Y -32.281,Z -68.498,A -90.000,B 90.000,C 0.000} C_DIS
LIN {X -57.949,Y -32.289,Z -68.326,A -90.000,B 90.000,C 0.000} C_DIS
LIN {X -57.879,Y -32.293,Z -68.078,A -90.000,B 90.000,C 0.000} C_DIS
LIN {X -57.798,Y -32.299,Z -67.815,A -90.000,B 90.000,C 0.000} C_DIS
LIN {X -57.786,Y -32.302,Z -67.781,A -90.000,B 90.000,C 0.000} C_DIS
LIN {X -57.693,Y -32.320,Z -67.533,A -90.000,B 90.000,C 0.000} C_DIS
LIN {X -57.592,Y -32.337,Z -67.279,A -90.000,B 90.000,C 0.000} C_DIS
LIN {X -57.538,Y -32.340,Z -67.152,A -90.000,B 90.000,C 0.000} C_DIS
LIN {X -57.477,Y -32.341,Z -67.023,A -90.000,B 90.000,C 0.000} C_DIS
LIN {X -57.441,Y -32.340,Z -66.952,A -90.000,B 90.000,C 0.000} C_DIS
LIN {X -57.188,Y -32.331,Z -66.464,A -90.000,B 90.000,C 0.000} C_DIS
LIN {X -57.154,Y -32.328,Z -66.376,A -90.000,B 90.000,C 0.000} C_DIS
LIN {X -57.108,Y -32.328,Z -66.262,A -90.000,B 90.000,C 0.000} C_DIS
LIN {X -57.028,Y -32.329,Z -66.076,A -90.000,B 90.000,C 0.000} C_DIS
LIN {X -56.954,Y -32.328,Z -65.919,A -90.000,B 90.000,C 0.000} C_DIS
LIN {X -56.885,Y -32.321,Z -65.782,A -90.000,B 90.000,C 0.000} C_DIS
LIN {X -56.619,Y -32.270,Z -65.311,A -90.000,B 90.000,C 0.000} C_DIS
LIN {X -56.475,Y -32.245,Z -65.080,A -90.000,B 90.000,C 0.000} C_DIS
LIN {X -56.381,Y -32.231,Z -64.938,A -90.000,B 90.000,C 0.000} C_DIS
LIN {X -56.283,Y -32.221,Z -64.802,A -90.000,B 90.000,C 0.000} C_DIS
LIN {X -56.169,Y -32.209,Z -64.649,A -90.000,B 90.000,C 0.000} C_DIS
LIN {X -56.041,Y -32.193,Z -64.493,A -90.000,B 90.000,C 0.000} C_DIS
LIN {X -55.835,Y -32.169,Z -64.257,A -90.000,B 90.000,C 0.000} C_DIS
LIN {X -55.665,Y -32.134,Z -64.076,A -90.000,B 90.000,C 0.000} C_DIS
LIN {X -55.069,Y -32.021,Z -63.487,A -90.000,B 90.000,C 0.000} C_DIS
LIN {X -54.796,Y -31.970,Z -63.217,A -90.000,B 90.000,C 0.000} C_DIS
LIN {X -54.438,Y -31.895,Z -62.867,A -90.000,B 90.000,C 0.000} C_DIS
LIN {X -54.342,Y -31.876,Z -62.778,A -90.000,B 90.000,C 0.000} C_DIS
LIN {X -54.195,Y -31.841,Z -62.649,A -90.000,B 90.000,C 0.000} C_DIS
LIN {X -54.070,Y -31.813,Z -62.548,A -90.000,B 90.000,C 0.000} C_DIS
LIN {X -53.843,Y -31.768,Z -62.374,A -90.000,B 90.000,C 0.000} C_DIS
LIN {X -53.566,Y -31.719,Z -62.183,A -90.000,B 90.000,C 0.000} C_DIS
LIN {X -53.420,Y -31.695,Z -62.083,A -90.000,B 90.000,C 0.000} C_DIS
LIN {X -53.263,Y -31.671,Z -61.983,A -90.000,B 90.000,C 0.000} C_DIS
LIN {X -53.145,Y -31.655,Z -61.912,A -90.000,B 90.000,C 0.000} C_DIS
LIN {X -52.918,Y -31.620,Z -61.766,A -90.000,B 90.000,C 0.000} C_DIS
LIN {X -52.239,Y -31.497,Z -61.340,A -90.000,B 90.000,C 0.000} C_DIS
LIN {X -51.997,Y -31.457,Z -61.198,A -90.000,B 90.000,C 0.000} C_DIS
LIN {X -51.481,Y -31.381,Z -60.914,A -90.000,B 90.000,C 0.000} C_DIS
LIN {X -51.267,Y -31.352,Z -60.802,A -90.000,B 90.000,C 0.000} C_DIS
LIN {X -51.188,Y -31.341,Z -60.763,A -90.000,B 90.000,C 0.000} C_DIS
LIN {X -50.935,Y -31.308,Z -60.645,A -90.000,B 90.000,C 0.000} C_DIS
LIN {X -50.935,Y -60.000,Z -60.645,A -90.000,B 90.000,C 0.000} C_DIS
LIN {X -60.567,Y -60.000,Z -76.632,A -90.000,B 90.000,C 0.000} C_DIS
LIN {X -60.567,Y -31.308,Z -76.632,A -90.000,B 90.000,C 0.000} C_DIS
LIN {X -60.569,Y -31.313,Z -76.571,A -90.000,B 90.000,C 0.000} C_DIS
LIN {X -60.578,Y -31.320,Z -76.450,A -90.000,B 90.000,C 0.000} C_DIS
LIN {X -60.593,Y -31.343,Z -76.112,A -90.000,B 90.000,C 0.000} C_DIS
LIN {X -60.603,Y -31.383,Z -75.473,A -90.000,B 90.000,C 0.000} C_DIS
LIN {X -60.609,Y -31.409,Z -75.020,A -90.000,B 90.000,C 0.000} C_DIS
LIN {X -60.625,Y -31.420,Z -74.764,A -90.000,B 90.000,C 0.000} C_DIS
LIN {X -60.634,Y -31.436,Z -74.445,A -90.000,B 90.000,C 0.000} C_DIS
LIN {X -60.633,Y -31.444,Z -74.303,A -90.000,B 90.000,C 0.000} C_DIS
LIN {X -60.623,Y -31.465,Z -73.973,A -90.000,B 90.000,C 0.000} C_DIS
LIN {X -60.607,Y -31.484,Z -73.685,A -90.000,B 90.000,C 0.000} C_DIS
LIN {X -60.572,Y -31.528,Z -73.126,A -90.000,B 90.000,C 0.000} C_DIS
LIN {X -60.578,Y -31.541,Z -72.896,A -90.000,B 90.000,C 0.000} C_DIS
LIN {X -60.575,Y -31.559,Z -72.624,A -90.000,B 90.000,C 0.000} C_DIS
LIN {X -60.563,Y -31.580,Z -72.364,A -90.000,B 90.000,C 0.000} C_DIS
LIN {X -60.535,Y -31.616,Z -71.933,A -90.000,B 90.000,C 0.000} C_DIS
LIN {X -60.518,Y -31.632,Z -71.760,A -90.000,B 90.000,C 0.000} C_DIS
LIN {X -60.493,Y -31.654,Z -71.538,A -90.000,B 90.000,C 0.000} C_DIS
LIN {X -60.407,Y -31.712,Z -70.949,A -90.000,B 90.000,C 0.000} C_DIS
LIN {X -60.391,Y -31.733,Z -70.694,A -90.000,B 90.000,C 0.000} C_DIS
LIN {X -60.381,Y -31.747,Z -70.553,A -90.000,B 90.000,C 0.000} C_DIS
LIN {X -60.371,Y -31.758,Z -70.422,A -90.000,B 90.000,C 0.000} C_DIS
LIN {X -60.351,Y -31.773,Z -70.246,A -90.000,B 90.000,C 0.000} C_DIS
LIN {X -60.290,Y -31.811,Z -69.822,A -90.000,B 90.000,C 0.000} C_DIS
LIN {X -60.266,Y -31.824,Z -69.681,A -90.000,B 90.000,C 0.000} C_DIS
LIN {X -60.237,Y -31.843,Z -69.528,A -90.000,B 90.000,C 0.000} C_DIS
LIN {X -60.228,Y -31.849,Z -69.480,A -90.000,B 90.000,C 0.000} C_DIS
LIN {X -60.185,Y -31.871,Z -69.293,A -90.000,B 90.000,C 0.000} C_DIS
LIN {X -60.130,Y -31.895,Z -69.069,A -90.000,B 90.000,C 0.000} C_DIS
LIN {X -60.045,Y -31.927,Z -68.744,A -90.000,B 90.000,C 0.000} C_DIS
LIN {X -60.002,Y -31.950,Z -68.459,A -90.000,B 90.000,C 0.000} C_DIS
LIN {X -59.956,Y -31.980,Z -68.206,A -90.000,B 90.000,C 0.000} C_DIS
LIN {X -59.919,Y -31.994,Z -68.047,A -90.000,B 90.000,C 0.000} C_DIS
LIN {X -59.852,Y -32.008,Z -67.779,A -90.000,B 90.000,C 0.000} C_DIS
LIN {X -59.762,Y -32.027,Z -67.458,A -90.000,B 90.000,C 0.000} C_DIS
LIN {X -59.696,Y -32.042,Z -67.241,A -90.000,B 90.000,C 0.000} C_DIS
LIN {X -59.645,Y -32.057,Z -67.085,A -90.000,B 90.000,C 0.000} C_DIS
LIN {X -59.560,Y -32.069,Z -66.861,A -90.000,B 90.000,C 0.000} C_DIS
LIN {X -59.506,Y -32.072,Z -66.723,A -90.000,B 90.000,C 0.000} C_DIS
LIN {X -59.385,Y -32.073,Z -66.430,A -90.000,B 90.000,C 0.000} C_DIS
LIN {X -59.318,Y -32.074,Z -66.280,A -90.000,B 90.000,C 0.000} C_DIS
LIN {X -59.209,Y -32.077,Z -66.055,A -90.000,B 90.000,C 0.000} C_DIS
LIN {X -59.050,Y -32.083,Z -65.745,A -90.000,B 90.000,C 0.000} C_DIS
LIN {X -59.003,Y -32.083,Z -65.654,A -90.000,B 90.000,C 0.000} C_DIS
LIN {X -58.971,Y -32.081,Z -65.575,A -90.000,B 90.000,C 0.000} C_DIS
LIN {X -58.917,Y -32.074,Z -65.447,A -90.000,B 90.000,C 0.000} C_DIS
LIN {X -58.819,Y -32.053,Z -65.228,A -90.000,B 90.000,C 0.000} C_DIS
LIN {X -58.727,Y -32.036,Z -65.040,A -90.000,B 90.000,C 0.000} C_DIS
LIN {X -58.658,Y -32.025,Z -64.905,A -90.000,B 90.000,C 0.000} C_DIS
LIN {X -58.369,Y -31.979,Z -64.386,A -90.000,B 90.000,C 0.000} C_DIS
LIN {X -58.311,Y -31.968,Z -64.288,A -90.000,B 90.000,C 0.000} C_DIS
LIN {X -58.166,Y -31.940,Z -64.056,A -90.000,B 90.000,C 0.000} C_DIS
LIN {X -58.088,Y -31.926,Z -63.938,A -90.000,B 90.000,C 0.000} C_DIS
LIN {X -57.997,Y -31.898,Z -63.808,A -90.000,B 90.000,C 0.000} C_DIS
LIN {X -57.875,Y -31.864,Z -63.644,A -90.000,B 90.000,C 0.000} C_DIS
LIN {X -57.759,Y -31.835,Z -63.495,A -90.000,B 90.000,C 0.000} C_DIS
LIN {X -57.659,Y -31.812,Z -63.374,A -90.000,B 90.000,C 0.000} C_DIS
LIN {X -57.518,Y -31.780,Z -63.209,A -90.000,B 90.000,C 0.000} C_DIS
LIN {X -57.264,Y -31.728,Z -62.928,A -90.000,B 90.000,C 0.000} C_DIS
LIN {X -57.048,Y -31.677,Z -62.704,A -90.000,B 90.000,C 0.000} C_DIS
LIN {X -56.817,Y -31.626,Z -62.478,A -90.000,B 90.000,C 0.000} C_DIS
LIN {X -56.337,Y -31.501,Z -62.017,A -90.000,B 90.000,C 0.000} C_DIS
LIN {X -55.843,Y -31.375,Z -61.542,A -90.000,B 90.000,C 0.000} C_DIS
LIN {X -55.727,Y -31.347,Z -61.436,A -90.000,B 90.000,C 0.000} C_DIS
LIN {X -55.582,Y -31.308,Z -61.310,A -90.000,B 90.000,C 0.000} C_DIS
LIN {X -55.582,Y -60.000,Z -61.310,A -90.000,B 90.000,C 0.000} C_DIS
LIN {X -62.424,Y -60.000,Z -71.138,A -90.000,B 90.000,C 0.000} C_DIS
LIN {X -62.424,Y -31.308,Z -71.138,A -90.000,B 90.000,C 0.000} C_DIS
LIN {X -62.396,Y -31.329,Z -70.948,A -90.000,B 90.000,C 0.000} C_DIS
LIN {X -62.381,Y -31.339,Z -70.843,A -90.000,B 90.000,C 0.000} C_DIS
LIN {X -62.363,Y -31.355,Z -70.714,A -90.000,B 90.000,C 0.000} C_DIS
LIN {X -62.341,Y -31.395,Z -70.366,A -90.000,B 90.000,C 0.000} C_DIS
LIN {X -62.326,Y -31.417,Z -70.174,A -90.000,B 90.000,C 0.000} C_DIS
LIN {X -62.307,Y -31.436,Z -70.004,A -90.000,B 90.000,C 0.000} C_DIS
LIN {X -62.284,Y -31.451,Z -69.836,A -90.000,B 90.000,C 0.000} C_DIS
LIN {X -62.233,Y -31.498,Z -69.466,A -90.000,B 90.000,C 0.000} C_DIS
LIN {X -62.197,Y -31.526,Z -69.249,A -90.000,B 90.000,C 0.000} C_DIS
LIN {X -62.147,Y -31.560,Z -68.994,A -90.000,B 90.000,C 0.000} C_DIS
LIN {X -62.088,Y -31.590,Z -68.744,A -90.000,B 90.000,C 0.000} C_DIS
LIN {X -62.075,Y -31.595,Z -68.691,A -90.000,B 90.000,C 0.000} C_DIS
LIN {X -61.982,Y -31.646,Z -68.321,A -90.000,B 90.000,C 0.000} C_DIS
LIN {X -61.947,Y -31.675,Z -68.081,A -90.000,B 90.000,C 0.000} C_DIS
LIN {X -61.893,Y -31.712,Z -67.785,A -90.000,B 90.000,C 0.000} C_DIS
LIN {X -61.861,Y -31.724,Z -67.647,A -90.000,B 90.000,C 0.000} C_DIS
LIN {X -61.848,Y -31.727,Z -67.591,A -90.000,B 90.000,C 0.000} C_DIS
LIN {X -61.758,Y -31.761,Z -67.226,A -90.000,B 90.000,C 0.000} C_DIS
LIN {X -61.651,Y -31.799,Z -66.842,A -90.000,B 90.000,C 0.000} C_DIS
LIN {X -61.601,Y -31.812,Z -66.677,A -90.000,B 90.000,C 0.000} C_DIS
LIN {X -61.547,Y -31.819,Z -66.512,A -90.000,B 90.000,C 0.000} C_DIS
LIN {X -61.497,Y -31.822,Z -66.369,A -90.000,B 90.000,C 0.000} C_DIS
LIN {X -61.460,Y -31.822,Z -66.272,A -90.000,B 90.000,C 0.000} C_DIS
LIN {X -61.340,Y -31.833,Z -65.962,A -90.000,B 90.000,C 0.000} C_DIS
LIN {X -61.260,Y -31.840,Z -65.767,A -90.000,B 90.000,C 0.000} C_DIS
LIN {X -61.176,Y -31.847,Z -65.567,A -90.000,B 90.000,C 0.000} C_DIS
LIN {X -61.107,Y -31.850,Z -65.415,A -90.000,B 90.000,C 0.000} C_DIS
LIN {X -61.025,Y -31.848,Z -65.246,A -90.000,B 90.000,C 0.000} C_DIS
LIN {X -60.974,Y -31.843,Z -65.144,A -90.000,B 90.000,C 0.000} C_DIS
LIN {X -60.807,Y -31.817,Z -64.828,A -90.000,B 90.000,C 0.000} C_DIS
LIN {X -60.734,Y -31.805,Z -64.655,A -90.000,B 90.000,C 0.000} C_DIS
LIN {X -60.608,Y -31.787,Z -64.376,A -90.000,B 90.000,C 0.000} C_DIS
LIN {X -60.504,Y -31.772,Z -64.161,A -90.000,B 90.000,C 0.000} C_DIS
LIN {X -60.432,Y -31.755,Z -64.023,A -90.000,B 90.000,C 0.000} C_DIS
LIN {X -60.236,Y -31.709,Z -63.671,A -90.000,B 90.000,C 0.000} C_DIS
LIN {X -60.086,Y -31.656,Z -63.414,A -90.000,B 90.000,C 0.000} C_DIS
LIN {X -59.979,Y -31.621,Z -63.240,A -90.000,B 90.000,C 0.000} C_DIS
LIN {X -59.873,Y -31.589,Z -63.075,A -90.000,B 90.000,C 0.000} C_DIS
LIN {X -59.713,Y -31.545,Z -62.836,A -90.000,B 90.000,C 0.000} C_DIS
LIN {X -59.607,Y -31.517,Z -62.685,A -90.000,B 90.000,C 0.000} C_DIS
LIN {X -59.418,Y -31.458,Z -62.437,A -90.000,B 90.000,C 0.000} C_DIS
LIN {X -59.310,Y -31.425,Z -62.300,A -90.000,B 90.000,C 0.000} C_DIS
LIN {X -59.231,Y -31.402,Z -62.207,A -90.000,B 90.000,C 0.000} C_DIS
LIN {X -59.005,Y -31.333,Z -61.948,A -90.000,B 90.000,C 0.000} C_DIS
LIN {X -58.916,Y -31.308,Z -61.852,A -90.000,B 90.000,C 0.000} C_DIS
LIN {X -58.668,Y -31.243,Z -61.590,A -90.000,B 90.000,C 0.000} C_DIS
LIN {X -58.446,Y -31.186,Z -61.366,A -90.000,B 90.000,C 0.000} C_DIS
LIN {X -58.250,Y -31.134,Z -61.178,A -90.000,B 90.000,C 0.000} C_DIS
LIN {X -58.160,Y -31.111,Z -61.098,A -90.000,B 90.000,C 0.000} C_DIS
LIN {X -57.999,Y -31.071,Z -60.962,A -90.000,B 90.000,C 0.000} C_DIS
LIN {X -57.862,Y -31.043,Z -60.860,A -90.000,B 90.000,C 0.000} C_DIS
LIN {X -57.773,Y -31.027,Z -60.804,A -90.000,B 90.000,C 0.000} C_DIS
LIN {X -57.697,Y -31.018,Z -60.766,A -90.000,B 90.000,C 0.000} C_DIS
LIN {X -57.653,Y -31.014,Z -60.750,A -90.000,B 90.000,C 0.000} C_DIS
LIN {X -57.596,Y -31.013,Z -60.739,A -90.000,B 90.000,C 0.000} C_DIS
LIN {X -57.565,Y -31.015,Z -60.741,A -90.000,B 90.000,C 0.000} C_DIS
LIN {X -57.551,Y -31.017,Z -60.745,A -90.000,B 90.000,C 0.000} C_DIS
LIN {X -57.527,Y -31.023,Z -60.757,A -90.000,B 90.000,C 0.000} C_DIS
LIN {X -57.508,Y -31.030,Z -60.777,A -90.000,B 90.000,C 0.000} C_DIS
LIN {X -57.494,Y -31.039,Z -60.802,A -90.000,B 90.000,C 0.000} C_DIS
LIN {X -57.484,Y -31.051,Z -60.834,A -90.000,B 90.000,C 0.000} C_DIS
LIN {X -57.479,Y -31.072,Z -60.894,A -90.000,B 90.000,C 0.000} C_DIS
LIN {X -57.483,Y -31.096,Z -60.968,A -90.000,B 90.000,C 0.000} C_DIS
LIN {X -57.491,Y -31.115,Z -61.024,A -90.000,B 90.000,C 0.000} C_DIS
LIN {X -57.520,Y -31.160,Z -61.153,A -90.000,B 90.000,C 0.000} C_DIS
LIN {X -57.565,Y -31.211,Z -61.304,A -90.000,B 90.000,C 0.000} C_DIS
LIN {X -57.626,Y -31.263,Z -61.474,A -90.000,B 90.000,C 0.000} C_DIS
LIN {X -57.701,Y -31.318,Z -61.663,A -90.000,B 90.000,C 0.000} C_DIS
LIN {X -57.839,Y -31.410,Z -61.979,A -90.000,B 90.000,C 0.000} C_DIS
LIN {X -57.947,Y -31.477,Z -62.210,A -90.000,B 90.000,C 0.000} C_DIS
LIN {X -58.068,Y -31.548,Z -62.455,A -90.000,B 90.000,C 0.000} C_DIS
LIN {X -58.132,Y -31.583,Z -62.582,A -90.000,B 90.000,C 0.000} C_DIS
LIN {X -58.269,Y -31.642,Z -62.846,A -90.000,B 90.000,C 0.000} C_DIS
LIN {X -58.416,Y -31.700,Z -63.121,A -90.000,B 90.000,C 0.000} C_DIS
LIN {X -58.738,Y -31.821,Z -63.699,A -90.000,B 90.000,C 0.000} C_DIS
LIN {X -58.911,Y -31.876,Z -64.000,A -90.000,B 90.000,C 0.000} C_DIS
LIN {X -59.091,Y -31.910,Z -64.307,A -90.000,B 90.000,C 0.000} C_DIS
LIN {X -59.278,Y -31.930,Z -64.619,A -90.000,B 90.000,C 0.000} C_DIS
LIN {X -59.668,Y -31.980,Z -65.252,A -90.000,B 90.000,C 0.000} C_DIS
LIN {X -59.870,Y -31.989,Z -65.571,A -90.000,B 90.000,C 0.000} C_DIS
LIN {X -60.283,Y -31.958,Z -66.206,A -90.000,B 90.000,C 0.000} C_DIS
LIN {X -60.493,Y -31.947,Z -66.521,A -90.000,B 90.000,C 0.000} C_DIS
LIN {X -60.704,Y -31.926,Z -66.831,A -90.000,B 90.000,C 0.000} C_DIS
LIN {X -60.916,Y -31.883,Z -67.136,A -90.000,B 90.000,C 0.000} C_DIS
LIN {X -61.127,Y -31.835,Z -67.434,A -90.000,B 90.000,C 0.000} C_DIS
LIN {X -61.443,Y -31.777,Z -67.867,A -90.000,B 90.000,C 0.000} C_DIS
LIN {X -61.547,Y -31.752,Z -68.007,A -90.000,B 90.000,C 0.000} C_DIS
LIN {X -61.650,Y -31.722,Z -68.144,A -90.000,B 90.000,C 0.000} C_DIS
LIN {X -61.957,Y -31.635,Z -68.538,A -90.000,B 90.000,C 0.000} C_DIS
LIN {X -62.254,Y -31.555,Z -68.903,A -90.000,B 90.000,C 0.000} C_DIS
LIN {X -62.350,Y -31.527,Z -69.018,A -90.000,B 90.000,C 0.000} C_DIS
LIN {X -62.540,Y -31.471,Z -69.235,A -90.000,B 90.000,C 0.000} C_DIS
LIN {X -62.723,Y -31.418,Z -69.436,A -90.000,B 90.000,C 0.000} C_DIS
LIN {X -62.899,Y -31.369,Z -69.619,A -90.000,B 90.000,C 0.000} C_DIS
LIN {X -63.068,Y -31.322,Z -69.783,A -90.000,B 90.000,C 0.000} C_DIS
LIN {X -63.149,Y -31.299,Z -69.857,A -90.000,B 90.000,C 0.000} C_DIS
LIN {X -63.304,Y -31.252,Z -69.990,A -90.000,B 90.000,C 0.000} C_DIS
LIN {X -63.451,Y -31.213,Z -70.101,A -90.000,B 90.000,C 0.000} C_DIS
LIN {X -63.587,Y -31.179,Z -70.187,A -90.000,B 90.000,C 0.000} C_DIS
LIN {X -63.682,Y -31.156,Z -70.236,A -90.000,B 90.000,C 0.000} C_DIS
LIN {X -63.770,Y -31.136,Z -70.271,A -90.000,B 90.000,C 0.000} C_DIS
LIN {X -63.825,Y -31.124,Z -70.285,A -90.000,B 90.000,C 0.000} C_DIS
LIN {X -63.877,Y -31.114,Z -70.293,A -90.000,B 90.000,C 0.000} C_DIS
LIN {X -63.949,Y -31.100,Z -70.292,A -90.000,B 90.000,C 0.000} C_DIS
LIN {X -63.993,Y -31.093,Z -70.282,A -90.000,B 90.000,C 0.000} C_DIS
LIN {X -64.014,Y -31.090,Z -70.274,A -90.000,B 90.000,C 0.000} C_DIS
LIN {X -64.052,Y -31.085,Z -70.253,A -90.000,B 90.000,C 0.000} C_DIS
LIN {X -64.070,Y -31.083,Z -70.239,A -90.000,B 90.000,C 0.000} C_DIS
LIN {X -64.104,Y -31.080,Z -70.207,A -90.000,B 90.000,C 0.000} C_DIS
LIN {X -64.119,Y -31.079,Z -70.187,A -90.000,B 90.000,C 0.000} C_DIS
LIN {X -64.146,Y -31.078,Z -70.143,A -90.000,B 90.000,C 0.000} C_DIS
LIN {X -64.170,Y -31.079,Z -70.090,A -90.000,B 90.000,C 0.000} C_DIS
LIN {X -64.190,Y -31.082,Z -70.029,A -90.000,B 90.000,C 0.000} C_DIS
LIN {X -64.212,Y -31.092,Z -69.922,A -90.000,B 90.000,C 0.000} C_DIS
LIN {X -64.222,Y -31.101,Z -69.840,A -90.000,B 90.000,C 0.000} C_DIS
LIN {X -64.227,Y -31.112,Z -69.749,A -90.000,B 90.000,C 0.000} C_DIS
LIN {X -64.228,Y -31.125,Z -69.649,A -90.000,B 90.000,C 0.000} C_DIS
LIN {X -64.225,Y -31.140,Z -69.540,A -90.000,B 90.000,C 0.000} C_DIS
LIN {X -64.211,Y -31.162,Z -69.359,A -90.000,B 90.000,C 0.000} C_DIS
LIN {X -64.196,Y -31.178,Z -69.226,A -90.000,B 90.000,C 0.000} C_DIS
LIN {X -64.176,Y -31.197,Z -69.084,A -90.000,B 90.000,C 0.000} C_DIS
LIN {X -64.122,Y -31.249,Z -68.770,A -90.000,B 90.000,C 0.000} C_DIS
LIN {X -64.047,Y -31.308,Z -68.415,A -90.000,B 90.000,C 0.000} C_DIS
LIN {X -64.012,Y -31.335,Z -68.259,A -90.000,B 90.000,C 0.000} C_DIS
LIN {X -63.923,Y -31.387,Z -67.902,A -90.000,B 90.000,C 0.000} C_DIS
LIN {X -63.891,Y -31.413,Z -67.693,A -90.000,B 90.000,C 0.000} C_DIS
LIN {X -63.838,Y -31.450,Z -67.403,A -90.000,B 90.000,C 0.000} C_DIS
LIN {X -63.771,Y -31.489,Z -67.095,A -90.000,B 90.000,C 0.000} C_DIS
LIN {X -63.720,Y -31.517,Z -66.884,A -90.000,B 90.000,C 0.000} C_DIS
LIN {X -63.661,Y -31.539,Z -66.652,A -90.000,B 90.000,C 0.000} C_DIS
LIN {X -63.582,Y -31.565,Z -66.371,A -90.000,B 90.000,C 0.000} C_DIS
LIN {X -63.487,Y -31.585,Z -66.052,A -90.000,B 90.000,C 0.000} C_DIS
LIN {X -63.422,Y -31.596,Z -65.852,A -90.000,B 90.000,C 0.000} C_DIS
LIN {X -63.353,Y -31.604,Z -65.657,A -90.000,B 90.000,C 0.000} C_DIS
LIN {X -63.197,Y -31.617,Z -65.250,A -90.000,B 90.000,C 0.000} C_DIS
LIN {X -63.155,Y -31.619,Z -65.147,A -90.000,B 90.000,C 0.000} C_DIS
LIN {X -63.088,Y -31.617,Z -64.987,A -90.000,B 90.000,C 0.000} C_DIS
LIN {X -62.984,Y -31.608,Z -64.748,A -90.000,B 90.000,C 0.000} C_DIS
LIN {X -62.889,Y -31.600,Z -64.542,A -90.000,B 90.000,C 0.000} C_DIS
LIN {X -62.719,Y -31.580,Z -64.201,A -90.000,B 90.000,C 0.000} C_DIS
LIN {X -62.608,Y -31.568,Z -63.989,A -90.000,B 90.000,C 0.000} C_DIS
LIN {X -62.565,Y -31.558,Z -63.889,A -90.000,B 90.000,C 0.000} C_DIS
LIN {X -62.396,Y -31.511,Z -63.523,A -90.000,B 90.000,C 0.000} C_DIS
LIN {X -62.346,Y -31.497,Z -63.421,A -90.000,B 90.000,C 0.000} C_DIS
LIN {X -62.204,Y -31.445,Z -63.147,A -90.000,B 90.000,C 0.000} C_DIS
LIN {X -61.906,Y -31.349,Z -62.625,A -90.000,B 90.000,C 0.000} C_DIS
LIN {X -61.820,Y -31.324,Z -62.473,A -90.000,B 90.000,C 0.000} C_DIS
LIN {X -61.782,Y -31.308,Z -62.412,A -90.000,B 90.000,C 0.000} C_DIS
LIN {X -61.555,Y -31.222,Z -62.043,A -90.000,B 90.000,C 0.000} C_DIS
LIN {X -61.275,Y -31.105,Z -61.593,A -90.000,B 90.000,C 0.000} C_DIS
LIN {X -61.201,Y -31.075,Z -61.480,A -90.000,B 90.000,C 0.000} C_DIS
LIN {X -61.234,Y -31.091,Z -61.539,A -90.000,B 90.000,C 0.000} C_DIS
LIN {X -61.416,Y -31.170,Z -61.839,A -90.000,B 90.000,C 0.000} C_DIS
LIN {X -61.732,Y -31.298,Z -62.344,A -90.000,B 90.000,C 0.000} C_DIS
LIN {X -61.931,Y -31.355,Z -62.657,A -90.000,B 90.000,C 0.000} C_DIS
LIN {X -62.391,Y -31.482,Z -63.371,A -90.000,B 90.000,C 0.000} C_DIS
LIN {X -62.646,Y -31.536,Z -63.759,A -90.000,B 90.000,C 0.000} C_DIS
LIN {X -63.048,Y -31.567,Z -64.359,A -90.000,B 90.000,C 0.000} C_DIS
LIN {X -63.186,Y -31.573,Z -64.561,A -90.000,B 90.000,C 0.000} C_DIS
LIN {X -63.463,Y -31.577,Z -64.963,A -90.000,B 90.000,C 0.000} C_DIS
LIN {X -63.602,Y -31.572,Z -65.161,A -90.000,B 90.000,C 0.000} C_DIS
LIN {X -63.879,Y -31.545,Z -65.547,A -90.000,B 90.000,C 0.000} C_DIS
LIN {X -64.150,Y -31.503,Z -65.914,A -90.000,B 90.000,C 0.000} C_DIS
LIN {X -64.413,Y -31.461,Z -66.256,A -90.000,B 90.000,C 0.000} C_DIS
LIN {X -64.539,Y -31.436,Z -66.415,A -90.000,B 90.000,C 0.000} C_DIS
LIN {X -64.662,Y -31.408,Z -66.565,A -90.000,B 90.000,C 0.000} C_DIS
LIN {X -64.781,Y -31.376,Z -66.706,A -90.000,B 90.000,C 0.000} C_DIS
LIN {X -64.951,Y -31.333,Z -66.897,A -90.000,B 90.000,C 0.000} C_DIS
LIN {X -65.109,Y -31.295,Z -67.062,A -90.000,B 90.000,C 0.000} C_DIS
LIN {X -65.254,Y -31.262,Z -67.197,A -90.000,B 90.000,C 0.000} C_DIS
LIN {X -65.342,Y -31.241,Z -67.270,A -90.000,B 90.000,C 0.000} C_DIS
LIN {X -65.423,Y -31.222,Z -67.327,A -90.000,B 90.000,C 0.000} C_DIS
LIN {X -65.461,Y -31.213,Z -67.350,A -90.000,B 90.000,C 0.000} C_DIS
LIN {X -65.531,Y -31.198,Z -67.383,A -90.000,B 90.000,C 0.000} C_DIS
LIN {X -65.563,Y -31.192,Z -67.393,A -90.000,B 90.000,C 0.000} C_DIS
LIN {X -65.607,Y -31.184,Z -67.400,A -90.000,B 90.000,C 0.000} C_DIS
LIN {X -65.633,Y -31.180,Z -67.399,A -90.000,B 90.000,C 0.000} C_DIS
LIN {X -65.657,Y -31.177,Z -67.393,A -90.000,B 90.000,C 0.000} C_DIS
LIN {X -65.689,Y -31.175,Z -67.375,A -90.000,B 90.000,C 0.000} C_DIS
LIN {X -65.708,Y -31.174,Z -67.358,A -90.000,B 90.000,C 0.000} C_DIS
LIN {X -65.730,Y -31.175,Z -67.321,A -90.000,B 90.000,C 0.000} C_DIS
LIN {X -65.743,Y -31.177,Z -67.291,A -90.000,B 90.000,C 0.000} C_DIS
LIN {X -65.756,Y -31.182,Z -67.235,A -90.000,B 90.000,C 0.000} C_DIS
LIN {X -65.761,Y -31.187,Z -67.191,A -90.000,B 90.000,C 0.000} C_DIS
LIN {X -65.764,Y -31.200,Z -67.086,A -90.000,B 90.000,C 0.000} C_DIS
LIN {X -65.755,Y -31.221,Z -66.957,A -90.000,B 90.000,C 0.000} C_DIS
LIN {X -65.746,Y -31.232,Z -66.885,A -90.000,B 90.000,C 0.000} C_DIS
LIN {X -65.719,Y -31.254,Z -66.720,A -90.000,B 90.000,C 0.000} C_DIS
LIN {X -65.655,Y -31.287,Z -66.426,A -90.000,B 90.000,C 0.000} C_DIS
LIN {X -65.596,Y -31.308,Z -66.198,A -90.000,B 90.000,C 0.000} C_DIS
LIN {X -65.531,Y -31.329,Z -65.960,A -90.000,B 90.000,C 0.000} C_DIS
LIN {X -65.483,Y -31.342,Z -65.791,A -90.000,B 90.000,C 0.000} C_DIS
LIN {X -65.358,Y -31.367,Z -65.376,A -90.000,B 90.000,C 0.000} C_DIS
LIN {X -65.294,Y -31.378,Z -65.183,A -90.000,B 90.000,C 0.000} C_DIS
LIN {X -65.236,Y -31.386,Z -65.020,A -90.000,B 90.000,C 0.000} C_DIS
LIN {X -65.167,Y -31.388,Z -64.836,A -90.000,B 90.000,C 0.000} C_DIS
LIN {X -65.058,Y -31.383,Z -64.556,A -90.000,B 90.000,C 0.000} C_DIS
LIN {X -64.912,Y -31.369,Z -64.205,A -90.000,B 90.000,C 0.000} C_DIS
LIN {X -64.789,Y -31.358,Z -63.922,A -90.000,B 90.000,C 0.000} C_DIS
LIN {X -64.691,Y -31.348,Z -63.711,A -90.000,B 90.000,C 0.000} C_DIS
LIN {X -64.523,Y -31.308,Z -63.380,A -90.000,B 90.000,C 0.000} C_DIS
LIN {X -64.523,Y -60.000,Z -63.380,A -90.000,B 90.000,C 0.000} C_DIS
LIN {X 4.584,Y -60.000,Z -172.867,A -90.000,B 90.000,C 0.000} C_DIS
LIN {X 4.584,Y -31.308,Z -172.867,A -90.000,B 90.000,C 0.000} C_DIS
LIN {X 4.795,Y -31.328,Z -172.576,A -90.000,B 90.000,C 0.000} C_DIS
LIN {X 5.833,Y -31.435,Z -171.206,A -90.000,B 90.000,C 0.000} C_DIS
LIN {X 5.947,Y -31.447,Z -171.057,A -90.000,B 90.000,C 0.000} C_DIS
LIN {X 6.064,Y -31.465,Z -170.898,A -90.000,B 90.000,C 0.000} C_DIS
LIN {X 6.269,Y -31.504,Z -170.616,A -90.000,B 90.000,C 0.000} C_DIS
LIN {X 6.946,Y -31.594,Z -169.421,A -90.000,B 90.000,C 0.000} C_DIS
LIN {X 7.178,Y -31.638,Z -169.001,A -90.000,B 90.000,C 0.000} C_DIS
LIN {X 7.338,Y -31.670,Z -168.720,A -90.000,B 90.000,C 0.000} C_DIS
LIN {X 7.608,Y -31.683,Z -167.872,A -90.000,B 90.000,C 0.000} C_DIS
LIN {X 7.663,Y -31.695,Z -167.684,A -90.000,B 90.000,C 0.000} C_DIS
LIN {X 7.918,Y -31.768,Z -166.798,A -90.000,B 90.000,C 0.000} C_DIS
LIN {X 7.944,Y -31.765,Z -166.398,A -90.000,B 90.000,C 0.000} C_DIS
LIN {X 7.936,Y -31.755,Z -166.214,A -90.000,B 90.000,C 0.000} C_DIS
LIN {X 7.912,Y -31.749,Z -165.806,A -90.000,B 90.000,C 0.000} C_DIS
LIN {X 7.896,Y -31.747,Z -165.460,A -90.000,B 90.000,C 0.000} C_DIS
LIN {X 7.823,Y -31.724,Z -164.918,A -90.000,B 90.000,C 0.000} C_DIS
LIN {X 7.758,Y -31.695,Z -164.417,A -90.000,B 90.000,C 0.000} C_DIS
LIN {X 7.744,Y -31.689,Z -164.357,A -90.000,B 90.000,C 0.000} C_DIS
LIN {X 7.591,Y -31.664,Z -163.777,A -90.000,B 90.000,C 0.000} C_DIS
LIN {X 7.515,Y -31.660,Z -163.503,A -90.000,B 90.000,C 0.000} C_DIS
LIN {X 7.185,Y -31.594,Z -162.769,A -90.000,B 90.000,C 0.000} C_DIS
LIN {X 7.123,Y -31.594,Z -162.642,A -90.000,B 90.000,C 0.000} C_DIS
LIN {X 7.026,Y -31.607,Z -162.462,A -90.000,B 90.000,C 0.000} C_DIS
LIN {X 6.994,Y -31.610,Z -162.405,A -90.000,B 90.000,C 0.000} C_DIS
LIN {X 6.956,Y -31.609,Z -162.358,A -90.000,B 90.000,C 0.000} C_DIS
LIN {X 6.213,Y -31.579,Z -161.444,A -90.000,B 90.000,C 0.000} C_DIS
LIN {X 6.139,Y -31.578,Z -161.349,A -90.000,B 90.000,C 0.000} C_DIS
LIN {X 5.763,Y -31.523,Z -161.028,A -90.000,B 90.000,C 0.000} C_DIS
LIN {X 5.214,Y -31.429,Z -160.545,A -90.000,B 90.000,C 0.000} C_DIS
LIN {X 5.166,Y -31.419,Z -160.502,A -90.000,B 90.000,C 0.000} C_DIS
LIN {X 4.984,Y -31.413,Z -160.358,A -90.000,B 90.000,C 0.000} C_DIS
LIN {X 4.411,Y -31.333,Z -160.035,A -90.000,B 90.000,C 0.000} C_DIS
LIN {X 4.227,Y -31.308,Z -159.928,A -90.000,B 90.000,C 0.000} C_DIS
LIN {X 4.227,Y -60.000,Z -159.928,A -90.000,B 90.000,C 0.000} C_DIS
LIN {X -99.827,Y -60.000,Z -243.561,A -90.000,B 90.000,C 0.000} C_DIS
LIN {X -99.827,Y -31.308,Z -243.561,A -90.000,B 90.000,C 0.000} C_DIS
LIN {X -99.575,Y -31.308,Z -243.372,A -90.000,B 90.000,C 0.000} C_DIS
LIN {X -99.213,Y -31.308,Z -243.118,A -90.000,B 90.000,C 0.000} C_DIS
LIN {X -93.942,Y -31.308,Z -239.465,A -90.000,B 90.000,C 0.000} C_DIS
LIN {X -91.480,Y -31.308,Z -237.722,A -90.000,B 90.000,C 0.000} C_DIS
LIN {X -87.487,Y -31.308,Z -235.121,A -90.000,B 90.000,C 0.000} C_DIS
LIN {X -83.358,Y -31.308,Z -232.376,A -90.000,B 90.000,C 0.000} C_DIS
LIN {X -80.799,Y -31.308,Z -230.806,A -90.000,B 90.000,C 0.000} C_DIS
LIN {X -74.941,Y -31.308,Z -227.169,A -90.000,B 90.000,C 0.000} C_DIS
LIN {X -74.553,Y -31.308,Z -226.942,A -90.000,B 90.000,C 0.000} C_DIS
LIN {X -71.717,Y -31.308,Z -225.317,A -90.000,B 90.000,C 0.000} C_DIS
LIN {X -66.272,Y -31.308,Z -222.244,A -90.000,B 90.000,C 0.000} C_DIS
LIN {X -65.976,Y -31.308,Z -222.084,A -90.000,B 90.000,C 0.000} C_DIS
LIN {X -64.509,Y -31.308,Z -221.303,A -90.000,B 90.000,C 0.000} C_DIS
LIN {X -59.150,Y -31.308,Z -218.478,A -90.000,B 90.000,C 0.000} C_DIS
LIN {X -57.474,Y -31.308,Z -217.600,A -90.000,B 90.000,C 0.000} C_DIS
LIN {X -53.054,Y -31.308,Z -215.345,A -90.000,B 90.000,C 0.000} C_DIS
LIN {X -49.513,Y -31.308,Z -213.553,A -90.000,B 90.000,C 0.000} C_DIS
LIN {X -47.411,Y -31.308,Z -212.485,A -90.000,B 90.000,C 0.000} C_DIS
LIN {X -42.479,Y -31.308,Z -209.987,A -90.000,B 90.000,C 0.000} C_DIS
LIN {X -41.301,Y -31.308,Z -209.360,A -90.000,B 90.000,C 0.000} C_DIS
LIN {X -37.087,Y -31.308,Z -207.129,A -90.000,B 90.000,C 0.000} C_DIS
LIN {X -35.525,Y -31.308,Z -206.247,A -90.000,B 90.000,C 0.000} C_DIS
LIN {X -32.834,Y -31.308,Z -204.741,A -90.000,B 90.000,C 0.000} C_DIS
LIN {X -32.329,Y -31.308,Z -204.452,A -90.000,B 90.000,C 0.000} C_DIS
LIN {X -29.229,Y -31.308,Z -202.576,A -90.000,B 90.000,C 0.000} C_DIS
LIN {X -28.263,Y -31.308,Z -201.981,A -90.000,B 90.000,C 0.000} C_DIS
LIN {X -25.910,Y -31.308,Z -200.441,A -90.000,B 90.000,C 0.000} C_DIS
LIN {X -24.830,Y -31.308,Z -199.722,A -90.000,B 90.000,C 0.000} C_DIS
LIN {X -23.382,Y -31.308,Z -198.701,A -90.000,B 90.000,C 0.000} C_DIS
LIN {X -21.579,Y -31.308,Z -197.442,A -90.000,B 90.000,C 0.000} C_DIS
LIN {X -19.910,Y -31.308,Z -196.187,A -90.000,B 90.000,C 0.000} C_DIS
LIN {X -18.260,Y -31.308,Z -194.954,A -90.000,B 90.000,C 0.000} C_DIS
LIN {X -16.433,Y -31.308,Z -193.498,A -90.000,B 90.000,C 0.000} C_DIS
LIN {X -14.935,Y -31.308,Z -192.301,A -90.000,B 90.000,C 0.000} C_DIS
LIN {X -12.818,Y -31.308,Z -190.525,A -90.000,B 90.000,C 0.000} C_DIS
LIN {X -11.560,Y -31.308,Z -189.457,A -90.000,B 90.000,C 0.000} C_DIS
LIN {X -10.151,Y -31.308,Z -188.200,A -90.000,B 90.000,C 0.000} C_DIS
LIN {X -8.112,Y -31.308,Z -186.420,A -90.000,B 90.000,C 0.000} C_DIS
LIN {X -6.764,Y -31.308,Z -185.155,A -90.000,B 90.000,C 0.000} C_DIS
LIN {X -4.538,Y -31.308,Z -183.135,A -90.000,B 90.000,C 0.000} C_DIS
LIN {X -2.154,Y -31.308,Z -180.765,A -90.000,B 90.000,C 0.000} C_DIS
LIN {X -1.165,Y -31.308,Z -179.823,A -90.000,B 90.000,C 0.000} C_DIS
LIN {X 1.414,Y -31.308,Z -177.048,A -90.000,B 90.000,C 0.000} C_DIS
LIN {X 1.637,Y -31.308,Z -176.821,A -90.000,B 90.000,C 0.000} C_DIS
LIN {X 1.773,Y -31.308,Z -176.673,A -90.000,B 90.000,C 0.000} C_DIS
LIN {X 3.284,Y -31.308,Z -174.811,A -90.000,B 90.000,C 0.000} C_DIS
LIN {X 4.114,Y -31.308,Z -173.658,A -90.000,B 90.000,C 0.000} C_DIS
LIN {X 4.286,Y -31.308,Z -173.397,A -90.000,B 90.000,C 0.000} C_DIS
LIN {X 4.755,Y -31.308,Z -172.563,A -90.000,B 90.000,C 0.000} C_DIS
LIN {X 5.448,Y -31.308,Z -171.369,A -90.000,B 90.000,C 0.000} C_DIS
LIN {X 5.746,Y -31.308,Z -170.743,A -90.000,B 90.000,C 0.000} C_DIS
LIN {X 6.077,Y -31.308,Z -169.886,A -90.000,B 90.000,C 0.000} C_DIS
LIN {X 6.202,Y -31.308,Z -169.436,A -90.000,B 90.000,C 0.000} C_DIS
LIN {X 6.231,Y -31.308,Z -169.338,A -90.000,B 90.000,C 0.000} C_DIS
LIN {X 6.526,Y -31.308,Z -168.333,A -90.000,B 90.000,C 0.000} C_DIS
LIN {X 6.585,Y -31.308,Z -168.145,A -90.000,B 90.000,C 0.000} C_DIS
LIN {X 6.763,Y -31.308,Z -167.196,A -90.000,B 90.000,C 0.000} C_DIS
LIN {X 6.806,Y -31.308,Z -166.703,A -90.000,B 90.000,C 0.000} C_DIS
LIN {X 6.796,Y -31.308,Z -166.287,A -90.000,B 90.000,C 0.000} C_DIS
LIN {X 6.805,Y -31.308,Z -165.593,A -90.000,B 90.000,C 0.000} C_DIS
LIN {X 6.843,Y -31.308,Z -164.847,A -90.000,B 90.000,C 0.000} C_DIS
LIN {X 6.540,Y -31.308,Z -162.887,A -90.000,B 90.000,C 0.000} C_DIS
LIN {X 6.281,Y -31.308,Z -162.532,A -90.000,B 90.000,C 0.000} C_DIS
LIN {X 5.088,Y -31.308,Z -160.779,A -90.000,B 90.000,C 0.000} C_DIS
LIN {X 4.951,Y -31.308,Z -160.549,A -90.000,B 90.000,C 0.000} C_DIS
LIN {X 3.619,Y -31.308,Z -159.405,A -90.000,B 90.000,C 0.000} C_DIS
LIN {X 2.946,Y -31.308,Z -158.812,A -90.000,B 90.000,C 0.000} C_DIS
LIN {X 2.120,Y -31.308,Z -158.332,A -90.000,B 90.000,C 0.000} C_DIS
LIN {X 0.771,Y -31.308,Z -157.536,A -90.000,B 90.000,C 0.000} C_DIS
LIN {X 0.455,Y -31.308,Z -157.340,A -90.000,B 90.000,C 0.000} C_DIS
LIN {X 0.115,Y -31.308,Z -157.181,A -90.000,B 90.000,C 0.000} C_DIS
LIN {X -0.287,Y -31.308,Z -156.990,A -90.000,B 90.000,C 0.000} C_DIS
LIN {X -1.484,Y -31.308,Z -156.397,A -90.000,B 90.000,C 0.000} C_DIS
LIN {X -2.086,Y -31.308,Z -156.094,A -90.000,B 90.000,C 0.000} C_DIS
LIN {X -2.389,Y -31.308,Z -155.921,A -90.000,B 90.000,C 0.000} C_DIS
LIN {X -2.801,Y -31.308,Z -155.750,A -90.000,B 90.000,C 0.000} C_DIS
LIN {X -5.335,Y -31.308,Z -154.622,A -90.000,B 90.000,C 0.000} C_DIS
LIN {X -5.766,Y -31.308,Z -154.408,A -90.000,B 90.000,C 0.000} C_DIS
LIN {X -7.865,Y -31.308,Z -153.479,A -90.000,B 90.000,C 0.000} C_DIS
LIN {X -8.533,Y -31.308,Z -153.181,A -90.000,B 90.000,C 0.000} C_DIS
LIN {X -8.984,Y -31.308,Z -152.942,A -90.000,B 90.000,C 0.000} C_DIS
LIN {X -9.455,Y -31.308,Z -152.704,A -90.000,B 90.000,C 0.000} C_DIS
LIN {X -11.735,Y -31.308,Z -151.551,A -90.000,B 90.000,C 0.000} C_DIS
LIN {X -12.162,Y -31.308,Z -151.339,A -90.000,B 90.000,C 0.000} C_DIS
LIN {X -14.638,Y -31.308,Z -149.890,A -90.000,B 90.000,C 0.000} C_DIS
LIN {X -15.436,Y -31.308,Z -149.454,A -90.000,B 90.000,C 0.000} C_DIS
LIN {X -15.833,Y -31.308,Z -149.227,A -90.000,B 90.000,C 0.000} C_DIS
LIN {X -16.722,Y -31.308,Z -148.626,A -90.000,B 90.000,C 0.000} C_DIS
LIN {X -19.431,Y -31.308,Z -146.886,A -90.000,B 90.000,C 0.000} C_DIS
LIN {X -19.729,Y -31.308,Z -146.672,A -90.000,B 90.000,C 0.000} C_DIS
LIN {X -20.442,Y -31.308,Z -146.135,A -90.000,B 90.000,C 0.000} C_DIS
LIN {X -22.217,Y -31.308,Z -144.777,A -90.000,B 90.000,C 0.000} C_DIS
LIN {X -23.314,Y -31.308,Z -143.968,A -90.000,B 90.000,C 0.000} C_DIS
LIN {X -23.533,Y -31.308,Z -143.792,A -90.000,B 90.000,C 0.000} C_DIS
LIN {X -25.794,Y -31.308,Z -141.819,A -90.000,B 90.000,C 0.000} C_DIS
LIN {X -26.401,Y -31.308,Z -141.277,A -90.000,B 90.000,C 0.000} C_DIS
LIN {X -26.790,Y -31.308,Z -140.938,A -90.000,B 90.000,C 0.000} C_DIS
LIN {X -27.070,Y -31.308,Z -140.690,A -90.000,B 90.000,C 0.000} C_DIS
LIN {X -28.225,Y -31.308,Z -139.478,A -90.000,B 90.000,C 0.000} C_DIS
LIN {X -30.156,Y -31.308,Z -137.510,A -90.000,B 90.000,C 0.000} C_DIS
LIN {X -30.443,Y -31.308,Z -137.197,A -90.000,B 90.000,C 0.000} C_DIS
LIN {X -30.481,Y -31.308,Z -137.153,A -90.000,B 90.000,C 0.000} C_DIS
LIN {X -30.719,Y -31.308,Z -136.854,A -90.000,B 90.000,C 0.000} C_DIS
LIN {X -32.174,Y -31.308,Z -134.982,A -90.000,B 90.000,C 0.000} C_DIS
LIN {X -33.015,Y -31.308,Z -133.919,A -90.000,B 90.000,C 0.000} C_DIS
LIN {X -33.303,Y -31.308,Z -133.532,A -90.000,B 90.000,C 0.000} C_DIS
LIN {X -34.002,Y -31.308,Z -132.431,A -90.000,B 90.000,C 0.000} C_DIS
LIN {X -35.362,Y -31.308,Z -130.297,A -90.000,B 90.000,C 0.000} C_DIS
LIN {X -35.608,Y -31.308,Z -129.882,A -90.000,B 90.000,C 0.000} C_DIS
LIN {X -36.051,Y -31.308,Z -128.992,A -90.000,B 90.000,C 0.000} C_DIS
LIN {X -37.254,Y -31.308,Z -126.560,A -90.000,B 90.000,C 0.000} C_DIS
LIN {X -37.390,Y -31.308,Z -126.264,A -90.000,B 90.000,C 0.000} C_DIS
LIN {X -37.447,Y -31.308,Z -126.120,A -90.000,B 90.000,C 0.000} C_DIS
LIN {X -37.938,Y -31.308,Z -124.825,A -90.000,B 90.000,C 0.000} C_DIS
LIN {X -38.779,Y -31.308,Z -122.559,A -90.000,B 90.000,C 0.000} C_DIS
LIN {X -38.906,Y -31.308,Z -122.100,A -90.000,B 90.000,C 0.000} C_DIS
LIN {X -39.339,Y -31.308,Z -120.432,A -90.000,B 90.000,C 0.000} C_DIS
LIN {X -39.814,Y -31.308,Z -118.658,A -90.000,B 90.000,C 0.000} C_DIS
LIN {X -39.880,Y -31.308,Z -118.355,A -90.000,B 90.000,C 0.000} C_DIS
LIN {X -40.327,Y -31.308,Z -115.652,A -90.000,B 90.000,C 0.000} C_DIS
LIN {X -40.516,Y -31.308,Z -114.550,A -90.000,B 90.000,C 0.000} C_DIS
LIN {X -40.573,Y -31.308,Z -114.086,A -90.000,B 90.000,C 0.000} C_DIS
LIN {X -40.607,Y -31.308,Z -113.673,A -90.000,B 90.000,C 0.000} C_DIS
LIN {X -40.790,Y -31.308,Z -111.746,A -90.000,B 90.000,C 0.000} C_DIS
LIN {X -40.864,Y -31.308,Z -111.070,A -90.000,B 90.000,C 0.000} C_DIS
LIN {X -40.882,Y -31.308,Z -110.934,A -90.000,B 90.000,C 0.000} C_DIS
LIN {X -40.995,Y -31.308,Z -110.247,A -90.000,B 90.000,C 0.000} C_DIS
LIN {X -41.145,Y -31.308,Z -109.731,A -90.000,B 90.000,C 0.000} C_DIS
LIN {X -41.521,Y -31.308,Z -108.924,A -90.000,B 90.000,C 0.000} C_DIS
LIN {X -41.586,Y -31.308,Z -108.797,A -90.000,B 90.000,C 0.000} C_DIS
LIN {X -42.302,Y -31.308,Z -107.662,A -90.000,B 90.000,C 0.000} C_DIS
LIN {X -42.411,Y -31.308,Z -107.478,A -90.000,B 90.000,C 0.000} C_DIS
LIN {X -43.633,Y -31.308,Z -105.743,A -90.000,B 90.000,C 0.000} C_DIS
LIN {X -44.767,Y -31.308,Z -104.231,A -90.000,B 90.000,C 0.000} C_DIS
LIN {X -45.699,Y -31.308,Z -103.108,A -90.000,B 90.000,C 0.000} C_DIS
LIN {X -46.219,Y -31.308,Z -102.430,A -90.000,B 90.000,C 0.000} C_DIS
LIN {X -47.664,Y -31.308,Z -100.675,A -90.000,B 90.000,C 0.000} C_DIS
LIN {X -47.812,Y -31.308,Z -100.488,A -90.000,B 90.000,C 0.000} C_DIS
LIN {X -49.089,Y -31.308,Z -98.781,A -90.000,B 90.000,C 0.000} C_DIS
LIN {X -49.447,Y -31.308,Z -98.274,A -90.000,B 90.000,C 0.000} C_DIS
LIN {X -49.750,Y -31.308,Z -97.839,A -90.000,B 90.000,C 0.000} C_DIS
LIN {X -50.098,Y -31.308,Z -97.351,A -90.000,B 90.000,C 0.000} C_DIS
LIN {X -51.015,Y -31.308,Z -95.946,A -90.000,B 90.000,C 0.000} C_DIS
LIN {X -52.161,Y -31.308,Z -94.181,A -90.000,B 90.000,C 0.000} C_DIS
LIN {X -52.950,Y -31.308,Z -92.925,A -90.000,B 90.000,C 0.000} C_DIS
LIN {X -53.809,Y -31.308,Z -91.479,A -90.000,B 90.000,C 0.000} C_DIS
LIN {X -54.164,Y -31.308,Z -90.800,A -90.000,B 90.000,C 0.000} C_DIS
LIN {X -55.774,Y -31.308,Z -87.673,A -90.000,B 90.000,C 0.000} C_DIS
LIN {X -56.575,Y -31.308,Z -86.205,A -90.000,B 90.000,C 0.000} C_DIS
LIN {X -57.025,Y -31.308,Z -85.150,A -90.000,B 90.000,C 0.000} C_DIS
LIN {X -57.266,Y -31.308,Z -84.553,A -90.000,B 90.000,C 0.000} C_DIS
LIN {X -57.829,Y -31.308,Z -83.370,A -90.000,B 90.000,C 0.000} C_DIS
LIN {X -58.323,Y -31.308,Z -82.364,A -90.000,B 90.000,C 0.000} C_DIS
LIN {X -58.473,Y -31.308,Z -81.954,A -90.000,B 90.000,C 0.000} C_DIS
LIN {X -58.664,Y -31.308,Z -81.397,A -90.000,B 90.000,C 0.000} C_DIS
LIN {X -59.066,Y -31.308,Z -80.434,A -90.000,B 90.000,C 0.000} C_DIS
LIN {X -59.461,Y -31.308,Z -79.524,A -90.000,B 90.000,C 0.000} C_DIS
LIN {X -59.613,Y -31.308,Z -79.140,A -90.000,B 90.000,C 0.000} C_DIS
LIN {X -59.849,Y -31.308,Z -78.490,A -90.000,B 90.000,C 0.000} C_DIS
LIN {X -60.058,Y -31.308,Z -77.994,A -90.000,B 90.000,C 0.000} C_DIS
LIN {X -60.170,Y -31.308,Z -77.738,A -90.000,B 90.000,C 0.000} C_DIS
LIN {X -60.514,Y -31.308,Z -76.785,A -90.000,B 90.000,C 0.000} C_DIS
LIN {X -60.780,Y -31.308,Z -76.006,A -90.000,B 90.000,C 0.000} C_DIS
LIN {X -60.891,Y -31.308,Z -75.638,A -90.000,B 90.000,C 0.000} C_DIS
LIN {X -61.159,Y -31.308,Z -74.641,A -90.000,B 90.000,C 0.000} C_DIS
LIN {X -61.188,Y -31.308,Z -74.527,A -90.000,B 90.000,C 0.000} C_DIS
LIN {X -61.449,Y -31.308,Z -73.634,A -90.000,B 90.000,C 0.000} C_DIS
LIN {X -61.525,Y -31.308,Z -73.409,A -90.000,B 90.000,C 0.000} C_DIS
LIN {X -61.730,Y -31.308,Z -72.783,A -90.000,B 90.000,C 0.000} C_DIS
LIN {X -61.912,Y -31.308,Z -72.345,A -90.000,B 90.000,C 0.000} C_DIS
LIN {X -62.091,Y -31.308,Z -71.836,A -90.000,B 90.000,C 0.000} C_DIS
LIN {X -62.459,Y -31.308,Z -71.065,A -90.000,B 90.000,C 0.000} C_DIS
LIN {X -62.535,Y -31.308,Z -70.855,A -90.000,B 90.000,C 0.000} C_DIS
LIN {X -62.977,Y -31.308,Z -70.023,A -90.000,B 90.000,C 0.000} C_DIS
LIN {X -63.104,Y -31.308,Z -69.816,A -90.000,B 90.000,C 0.000} C_DIS
LIN {X -63.485,Y -31.308,Z -69.146,A -90.000,B 90.000,C 0.000} C_DIS
LIN {X -63.744,Y -31.308,Z -68.811,A -90.000,B 90.000,C 0.000} C_DIS
LIN {X -64.290,Y -31.308,Z -68.097,A -90.000,B 90.000,C 0.000} C_DIS
LIN {X -64.812,Y -31.308,Z -67.311,A -90.000,B 90.000,C 0.000} C_DIS
LIN {X -65.600,Y -31.308,Z -66.193,A -90.000,B 90.000,C 0.000} C_DIS
LIN {X -65.729,Y -31.308,Z -65.866,A -90.000,B 90.000,C 0.000} C_DIS
LIN {X -65.788,Y -31.308,Z -65.697,A -90.000,B 90.000,C 0.000} C_DIS
LIN {X -65.905,Y -31.308,Z -65.124,A -90.000,B 90.000,C 0.000} C_DIS
LIN {X -65.915,Y -31.308,Z -64.945,A -90.000,B 90.000,C 0.000} C_DIS
LIN {X -65.877,Y -31.308,Z -64.770,A -90.000,B 90.000,C 0.000} C_DIS
LIN {X -65.633,Y -31.308,Z -64.317,A -90.000,B 90.000,C 0.000} C_DIS
LIN {X -65.196,Y -31.308,Z -63.796,A -90.000,B 90.000,C 0.000} C_DIS
LIN {X -65.070,Y -31.308,Z -63.668,A -90.000,B 90.000,C 0.000} C_DIS
LIN {X -64.914,Y -31.308,Z -63.580,A -90.000,B 90.000,C 0.000} C_DIS
LIN {X -64.529,Y -31.308,Z -63.383,A -90.000,B 90.000,C 0.000} C_DIS
LIN {X -64.365,Y -31.308,Z -63.303,A -90.000,B 90.000,C 0.000} C_DIS
LIN {X -64.168,Y -31.308,Z -63.212,A -90.000,B 90.000,C 0.000} C_DIS
LIN {X -63.463,Y -31.308,Z -62.974,A -90.000,B 90.000,C 0.000} C_DIS
LIN {X -61.984,Y -31.308,Z -62.458,A -90.000,B 90.000,C 0.000} C_DIS
LIN {X -61.243,Y -31.308,Z -62.289,A -90.000,B 90.000,C 0.000} C_DIS
LIN {X -60.368,Y -31.308,Z -62.112,A -90.000,B 90.000,C 0.000} C_DIS
LIN {X -58.313,Y -31.308,Z -61.744,A -90.000,B 90.000,C 0.000} C_DIS
LIN {X -56.302,Y -31.308,Z -61.407,A -90.000,B 90.000,C 0.000} C_DIS
LIN {X -55.223,Y -31.308,Z -61.261,A -90.000,B 90.000,C 0.000} C_DIS
LIN {X -53.241,Y -31.308,Z -60.986,A -90.000,B 90.000,C 0.000} C_DIS
LIN {X -52.164,Y -31.308,Z -60.830,A -90.000,B 90.000,C 0.000} C_DIS
LIN {X -51.724,Y -31.308,Z -60.760,A -90.000,B 90.000,C 0.000} C_DIS
LIN {X -49.238,Y -31.308,Z -60.399,A -90.000,B 90.000,C 0.000} C_DIS
LIN {X -47.905,Y -31.308,Z -60.180,A -90.000,B 90.000,C 0.000} C_DIS
LIN {X -46.687,Y -31.308,Z -59.951,A -90.000,B 90.000,C 0.000} C_DIS
LIN {X -44.734,Y -31.308,Z -59.652,A -90.000,B 90.000,C 0.000} C_DIS
LIN {X -44.610,Y -31.308,Z -59.632,A -90.000,B 90.000,C 0.000} C_DIS
LIN {X -44.252,Y -31.308,Z -59.593,A -90.000,B 90.000,C 0.000} C_DIS
LIN {X -43.942,Y -31.308,Z -59.571,A -90.000,B 90.000,C 0.000} C_DIS
LIN {X -42.642,Y -31.308,Z -59.462,A -90.000,B 90.000,C 0.000} C_DIS
LIN {X -42.144,Y -31.308,Z -59.446,A -90.000,B 90.000,C 0.000} C_DIS
LIN {X -41.947,Y -31.308,Z -59.432,A -90.000,B 90.000,C 0.000} C_DIS
LIN {X -40.265,Y -31.308,Z -59.545,A -90.000,B 90.000,C 0.000} C_DIS
LIN {X -39.928,Y -31.308,Z -59.558,A -90.000,B 90.000,C 0.000} C_DIS
LIN {X -39.115,Y -31.308,Z -59.610,A -90.000,B 90.000,C 0.000} C_DIS
LIN {X -38.776,Y -31.308,Z -59.636,A -90.000,B 90.000,C 0.000} C_DIS
LIN {X -38.297,Y -31.308,Z -59.719,A -90.000,B 90.000,C 0.000} C_DIS
LIN {X -37.852,Y -31.308,Z -59.795,A -90.000,B 90.000,C 0.000} C_DIS
LIN {X -37.480,Y -31.308,Z -59.865,A -90.000,B 90.000,C 0.000} C_DIS
LIN {X -36.152,Y -31.308,Z -60.135,A -90.000,B 90.000,C 0.000} C_DIS
LIN {X -34.648,Y -31.308,Z -60.415,A -90.000,B 90.000,C 0.000} C_DIS
LIN {X -32.599,Y -31.308,Z -60.875,A -90.000,B 90.000,C 0.000} C_DIS
LIN {X -29.858,Y -31.308,Z -61.514,A -90.000,B 90.000,C 0.000} C_DIS
LIN {X -27.887,Y -31.308,Z -62.000,A -90.000,B 90.000,C 0.000} C_DIS
LIN {X -27.354,Y -31.308,Z -62.123,A -90.000,B 90.000,C 0.000} C_DIS
LIN {X -26.774,Y -31.308,Z -62.270,A -90.000,B 90.000,C 0.000} C_DIS
LIN {X -25.336,Y -31.308,Z -62.576,A -90.000,B 90.000,C 0.000} C_DIS
LIN {X -24.043,Y -31.308,Z -62.746,A -90.000,B 90.000,C 0.000} C_DIS
LIN {X -23.840,Y -31.308,Z -62.782,A -90.000,B 90.000,C 0.000} C_DIS
LIN {X -23.492,Y -31.308,Z -62.735,A -90.000,B 90.000,C 0.000} C_DIS
LIN {X -23.168,Y -31.308,Z -62.710,A -90.000,B 90.000,C 0.000} C_DIS
LIN {X -23.098,Y -31.308,Z -62.675,A -90.000,B 90.000,C 0.000} C_DIS
LIN {X -22.998,Y -31.308,Z -62.458,A -90.000,B 90.000,C 0.000} C_DIS
LIN {X -22.822,Y -31.308,Z -62.116,A -90.000,B 90.000,C 0.000} C_DIS
LIN {X -22.588,Y -31.308,Z -61.774,A -90.000,B 90.000,C 0.000} C_DIS
LIN {X -22.548,Y -31.308,Z -61.724,A -90.000,B 90.000,C 0.000} C_DIS
LIN {X -22.195,Y -31.308,Z -61.317,A -90.000,B 90.000,C 0.000} C_DIS
LIN {X -22.067,Y -31.308,Z -61.165,A -90.000,B 90.000,C 0.000} C_DIS
LIN {X -21.801,Y -31.308,Z -60.863,A -90.000,B 90.000,C 0.000} C_DIS
LIN {X -21.499,Y -31.308,Z -60.596,A -90.000,B 90.000,C 0.000} C_DIS
LIN {X -21.306,Y -31.308,Z -60.444,A -90.000,B 90.000,C 0.000} C_DIS
LIN {X -20.736,Y -31.308,Z -60.024,A -90.000,B 90.000,C 0.000} C_DIS
LIN {X -20.567,Y -31.308,Z -59.901,A -90.000,B 90.000,C 0.000} C_DIS
LIN {X -20.386,Y -31.308,Z -59.774,A -90.000,B 90.000,C 0.000} C_DIS
LIN {X -20.227,Y -31.308,Z -59.665,A -90.000,B 90.000,C 0.000} C_DIS
LIN {X -20.033,Y -31.308,Z -59.560,A -90.000,B 90.000,C 0.000} C_DIS
LIN {X -19.367,Y -31.308,Z -59.220,A -90.000,B 90.000,C 0.000} C_DIS
LIN {X -18.876,Y -31.308,Z -59.005,A -90.000,B 90.000,C 0.000} C_DIS
LIN {X -18.606,Y -31.308,Z -58.897,A -90.000,B 90.000,C 0.000} C_DIS
LIN {X -18.102,Y -31.308,Z -58.713,A -90.000,B 90.000,C 0.000} C_DIS
LIN {X -17.127,Y -31.308,Z -58.363,A -90.000,B 90.000,C 0.000} C_DIS
LIN {X -16.760,Y -31.308,Z -58.230,A -90.000,B 90.000,C 0.000} C_DIS
LIN {X -16.160,Y -31.308,Z -58.016,A -90.000,B 90.000,C 0.000} C_DIS
LIN {X -16.134,Y -31.308,Z -58.008,A -90.000,B 90.000,C 0.000} C_DIS
LIN {X -15.240,Y -31.308,Z -57.799,A -90.000,B 90.000,C 0.000} C_DIS
LIN {X -14.869,Y -31.308,Z -57.720,A -90.000,B 90.000,C 0.000} C_DIS
LIN {X -14.102,Y -31.308,Z -57.623,A -90.000,B 90.000,C 0.000} C_DIS
LIN {X -13.846,Y -31.308,Z -57.602,A -90.000,B 90.000,C 0.000} C_DIS
LIN {X -13.507,Y -31.308,Z -57.580,A -90.000,B 90.000,C 0.000} C_DIS
LIN {X -12.403,Y -31.308,Z -57.518,A -90.000,B 90.000,C 0.000} C_DIS
LIN {X -11.812,Y -31.308,Z -57.508,A -90.000,B 90.000,C 0.000} C_DIS
LIN {X -11.151,Y -31.308,Z -57.539,A -90.000,B 90.000,C 0.000} C_DIS
LIN {X -10.801,Y -31.308,Z -57.566,A -90.000,B 90.000,C 0.000} C_DIS
LIN {X -9.598,Y -31.308,Z -57.714,A -90.000,B 90.000,C 0.000} C_DIS
LIN {X -8.078,Y -31.308,Z -57.994,A -90.000,B 90.000,C 0.000} C_DIS
LIN {X -7.367,Y -31.308,Z -58.135,A -90.000,B 90.000,C 0.000} C_DIS
LIN {X -6.983,Y -31.308,Z -58.222,A -90.000,B 90.000,C 0.000} C_DIS
LIN {X -5.016,Y -31.308,Z -58.720,A -90.000,B 90.000,C 0.000} C_DIS
LIN {X -4.078,Y -31.308,Z -58.924,A -90.000,B 90.000,C 0.000} C_DIS
LIN {X -2.229,Y -31.308,Z -59.420,A -90.000,B 90.000,C 0.000} C_DIS
LIN {X -1.460,Y -31.308,Z -59.574,A -90.000,B 90.000,C 0.000} C_DIS
LIN {X 0.645,Y -31.308,Z -60.096,A -90.000,B 90.000,C 0.000} C_DIS
LIN {X 2.657,Y -31.308,Z -60.466,A -90.000,B 90.000,C 0.000} C_DIS
LIN {X 3.107,Y -31.308,Z -60.538,A -90.000,B 90.000,C 0.000} C_DIS
LIN {X 3.905,Y -31.308,Z -60.649,A -90.000,B 90.000,C 0.000} C_DIS
LIN {X 5.299,Y -31.308,Z -60.831,A -90.000,B 90.000,C 0.000} C_DIS
LIN {X 5.854,Y -31.308,Z -60.875,A -90.000,B 90.000,C 0.000} C_DIS
LIN {X 7.358,Y -31.308,Z -60.987,A -90.000,B 90.000,C 0.000} C_DIS
LIN {X 8.287,Y -31.308,Z -60.996,A -90.000,B 90.000,C 0.000} C_DIS
LIN {X 8.812,Y -31.308,Z -61.002,A -90.000,B 90.000,C 0.000} C_DIS
LIN {X 9.901,Y -31.308,Z -60.914,A -90.000,B 90.000,C 0.000} C_DIS
LIN {X 10.016,Y -31.308,Z -60.906,A -90.000,B 90.000,C 0.000} C_DIS
LIN {X 10.940,Y -31.308,Z -60.741,A -90.000,B 90.000,C 0.000} C_DIS
LIN {X 11.664,Y -31.308,Z -60.539,A -90.000,B 90.000,C 0.000} C_DIS
LIN {X 12.035,Y -31.308,Z -60.400,A -90.000,B 90.000,C 0.000} C_DIS
LIN {X 12.492,Y -31.308,Z -60.200,A -90.000,B 90.000,C 0.000} C_DIS
LIN {X 12.681,Y -31.308,Z -60.110,A -90.000,B 90.000,C 0.000} C_DIS
LIN {X 13.337,Y -31.308,Z -59.826,A -90.000,B 90.000,C 0.000} C_DIS
LIN {X 13.396,Y -31.308,Z -59.798,A -90.000,B 90.000,C 0.000} C_DIS
LIN {X 13.793,Y -31.308,Z -59.642,A -90.000,B 90.000,C 0.000} C_DIS
LIN {X 13.973,Y -31.308,Z -59.581,A -90.000,B 90.000,C 0.000} C_DIS
LIN {X 14.443,Y -31.308,Z -59.442,A -90.000,B 90.000,C 0.000} C_DIS
LIN {X 14.839,Y -31.308,Z -59.337,A -90.000,B 90.000,C 0.000} C_DIS
LIN {X 15.258,Y -31.308,Z -59.278,A -90.000,B 90.000,C 0.000} C_DIS
LIN {X 15.325,Y -31.308,Z -59.275,A -90.000,B 90.000,C 0.000} C_DIS
LIN {X 15.891,Y -31.308,Z -59.203,A -90.000,B 90.000,C 0.000} C_DIS
LIN {X 16.314,Y -31.308,Z -59.193,A -90.000,B 90.000,C 0.000} C_DIS
LIN {X 16.736,Y -31.308,Z -59.233,A -90.000,B 90.000,C 0.000} C_DIS
LIN {X 16.863,Y -31.308,Z -59.256,A -90.000,B 90.000,C 0.000} C_DIS
LIN {X 17.361,Y -31.308,Z -59.305,A -90.000,B 90.000,C 0.000} C_DIS
LIN {X 17.775,Y -31.308,Z -59.394,A -90.000,B 90.000,C 0.000} C_DIS
LIN {X 17.910,Y -31.308,Z -59.435,A -90.000,B 90.000,C 0.000} C_DIS
LIN {X 18.024,Y -31.308,Z -59.460,A -90.000,B 90.000,C 0.000} C_DIS
LIN {X 18.048,Y -31.308,Z -59.449,A -90.000,B 90.000,C 0.000} C_DIS
LIN {X 18.352,Y -31.308,Z -59.338,A -90.000,B 90.000,C 0.000} C_DIS
LIN {X 18.639,Y -31.308,Z -59.247,A -90.000,B 90.000,C 0.000} C_DIS
LIN {X 18.850,Y -31.308,Z -59.187,A -90.000,B 90.000,C 0.000} C_DIS
LIN {X 18.991,Y -31.308,Z -59.120,A -90.000,B 90.000,C 0.000} C_DIS
LIN {X 19.138,Y -31.308,Z -59.065,A -90.000,B 90.000,C 0.000} C_DIS
LIN {X 19.566,Y -31.308,Z -58.909,A -90.000,B 90.000,C 0.000} C_DIS
LIN {X 19.922,Y -31.308,Z -58.810,A -90.000,B 90.000,C 0.000} C_DIS
LIN {X 20.355,Y -31.308,Z -58.728,A -90.000,B 90.000,C 0.000} C_DIS
LIN {X 20.490,Y -31.308,Z -58.713,A -90.000,B 90.000,C 0.000} C_DIS
LIN {X 20.929,Y -31.308,Z -58.681,A -90.000,B 90.000,C 0.000} C_DIS
LIN {X 21.370,Y -31.308,Z -58.698,A -90.000,B 90.000,C 0.000} C_DIS
LIN {X 21.806,Y -31.308,Z -58.766,A -90.000,B 90.000,C 0.000} C_DIS
LIN {X 21.864,Y -31.308,Z -58.782,A -90.000,B 90.000,C 0.000} C_DIS
LIN {X 22.414,Y -31.308,Z -58.416,A -90.000,B 90.000,C 0.000} C_DIS
LIN {X 23.005,Y -31.308,Z -58.058,A -90.000,B 90.000,C 0.000} C_DIS
LIN {X 23.637,Y -31.308,Z -57.711,A -90.000,B 90.000,C 0.000} C_DIS
LIN {X 23.962,Y -31.308,Z -57.535,A -90.000,B 90.000,C 0.000} C_DIS
LIN {X 24.615,Y -31.308,Z -57.212,A -90.000,B 90.000,C 0.000} C_DIS
LIN {X 24.839,Y -31.308,Z -57.112,A -90.000,B 90.000,C 0.000} C_DIS
LIN {X 24.809,Y -31.308,Z -56.780,A -90.000,B 90.000,C 0.000} C_DIS
LIN {X 24.820,Y -31.308,Z -56.339,A -90.000,B 90.000,C 0.000} C_DIS
LIN {X 24.881,Y -31.308,Z -55.897,A -90.000,B 90.000,C 0.000} C_DIS
LIN {X 24.912,Y -31.308,Z -55.776,A -90.000,B 90.000,C 0.000} C_DIS
LIN {X 24.989,Y -31.308,Z -55.476,A -90.000,B 90.000,C 0.000} C_DIS
LIN {X 25.146,Y -31.308,Z -55.064,A -90.000,B 90.000,C 0.000} C_DIS
LIN {X 25.168,Y -31.308,Z -55.014,A -90.000,B 90.000,C 0.000} C_DIS
LIN {X 25.200,Y -31.308,Z -54.932,A -90.000,B 90.000,C 0.000} C_DIS
LIN {X 25.400,Y -31.308,Z -54.545,A -90.000,B 90.000,C 0.000} C_DIS
LIN {X 25.651,Y -31.308,Z -54.156,A -90.000,B 90.000,C 0.000} C_DIS
LIN {X 25.937,Y -31.308,Z -53.797,A -90.000,B 90.000,C 0.000} C_DIS
LIN {X 26.181,Y -31.308,Z -53.551,A -90.000,B 90.000,C 0.000} C_DIS
LIN {X 26.216,Y -31.308,Z -53.512,A -90.000,B 90.000,C 0.000} C_DIS
LIN {X 26.564,Y -31.308,Z -53.200,A -90.000,B 90.000,C 0.000} C_DIS
LIN {X 26.944,Y -31.308,Z -52.928,A -90.000,B 90.000,C 0.000} C_DIS
LIN {X 27.051,Y -31.308,Z -52.860,A -90.000,B 90.000,C 0.000} C_DIS
LIN {X 27.445,Y -31.308,Z -52.634,A -90.000,B 90.000,C 0.000} C_DIS
LIN {X 27.600,Y -31.308,Z -52.554,A -90.000,B 90.000,C 0.000} C_DIS
LIN {X 27.621,Y -31.308,Z -52.218,A -90.000,B 90.000,C 0.000} C_DIS
LIN {X 27.675,Y -31.308,Z -51.810,A -90.000,B 90.000,C 0.000} C_DIS
LIN {X 27.707,Y -31.308,Z -51.648,A -90.000,B 90.000,C 0.000} C_DIS
LIN {X 27.919,Y -31.308,Z -50.809,A -90.000,B 90.000,C 0.000} C_DIS
LIN {X 28.071,Y -31.308,Z -50.414,A -90.000,B 90.000,C 0.000} C_DIS
LIN {X 28.124,Y -31.308,Z -50.288,A -90.000,B 90.000,C 0.000} C_DIS
LIN {X 28.321,Y -31.308,Z -49.832,A -90.000,B 90.000,C 0.000} C_DIS
LIN {X 28.560,Y -31.308,Z -49.383,A -90.000,B 90.000,C 0.000} C_DIS
LIN {X 28.715,Y -31.308,Z -49.146,A -90.000,B 90.000,C 0.000} C_DIS
LIN {X 28.914,Y -31.308,Z -48.822,A -90.000,B 90.000,C 0.000} C_DIS
LIN {X 28.925,Y -31.308,Z -48.806,A -90.000,B 90.000,C 0.000} C_DIS
LIN {X 29.160,Y -31.308,Z -48.456,A -90.000,B 90.000,C 0.000} C_DIS
LIN {X 29.445,Y -31.308,Z -48.120,A -90.000,B 90.000,C 0.000} C_DIS
LIN {X 29.717,Y -31.308,Z -47.862,A -90.000,B 90.000,C 0.000} C_DIS
LIN {X 29.950,Y -31.308,Z -47.616,A -90.000,B 90.000,C 0.000} C_DIS
LIN {X 30.272,Y -31.308,Z -47.315,A -90.000,B 90.000,C 0.000} C_DIS
LIN {X 30.703,Y -31.308,Z -46.988,A -90.000,B 90.000,C 0.000} C_DIS
LIN {X 31.086,Y -31.308,Z -46.742,A -90.000,B 90.000,C 0.000} C_DIS
LIN {X 31.814,Y -31.308,Z -46.346,A -90.000,B 90.000,C 0.000} C_DIS
LIN {X 32.223,Y -31.308,Z -46.144,A -90.000,B 90.000,C 0.000} C_DIS
LIN {X 32.650,Y -31.308,Z -45.988,A -90.000,B 90.000,C 0.000} C_DIS
LIN {X 33.167,Y -31.308,Z -45.850,A -90.000,B 90.000,C 0.000} C_DIS
LIN {X 33.626,Y -31.308,Z -45.760,A -90.000,B 90.000,C 0.000} C_DIS
LIN {X 33.919,Y -31.308,Z -45.712,A -90.000,B 90.000,C 0.000} C_DIS
LIN {X 34.631,Y -31.308,Z -45.571,A -90.000,B 90.000,C 0.000} C_DIS
LIN {X 35.096,Y -31.308,Z -45.530,A -90.000,B 90.000,C 0.000} C_DIS
LIN {X 35.648,Y -31.308,Z -45.499,A -90.000,B 90.000,C 0.000} C_DIS
LIN {X 36.350,Y -31.308,Z -45.521,A -90.000,B 90.000,C 0.000} C_DIS
LIN {X 36.826,Y -31.308,Z -45.544,A -90.000,B 90.000,C 0.000} C_DIS
LIN {X 37.169,Y -31.308,Z -45.573,A -90.000,B 90.000,C 0.000} C_DIS
LIN {X 37.452,Y -31.308,Z -45.602,A -90.000,B 90.000,C 0.000} C_DIS
LIN {X 37.784,Y -31.308,Z -45.653,A -90.000,B 90.000,C 0.000} C_DIS
LIN {X 38.972,Y -31.308,Z -45.829,A -90.000,B 90.000,C 0.000} C_DIS
LIN {X 40.015,Y -31.308,Z -45.952,A -90.000,B 90.000,C 0.000} C_DIS
LIN {X 40.613,Y -31.308,Z -45.957,A -90.000,B 90.000,C 0.000} C_DIS
LIN {X 41.296,Y -31.308,Z -45.823,A -90.000,B 90.000,C 0.000} C_DIS
LIN {X 42.363,Y -31.308,Z -45.514,A -90.000,B 90.000,C 0.000} C_DIS
LIN {X 42.920,Y -31.308,Z -45.345,A -90.000,B 90.000,C 0.000} C_DIS
LIN {X 44.449,Y -31.308,Z -44.938,A -90.000,B 90.000,C 0.000} C_DIS
LIN {X 44.592,Y -31.308,Z -44.895,A -90.000,B 90.000,C 0.000} C_DIS
LIN {X 45.025,Y -31.308,Z -44.813,A -90.000,B 90.000,C 0.000} C_DIS
LIN {X 45.347,Y -31.308,Z -44.768,A -90.000,B 90.000,C 0.000} C_DIS
LIN {X 46.198,Y -31.308,Z -44.707,A -90.000,B 90.000,C 0.000} C_DIS
LIN {X 46.842,Y -31.308,Z -44.667,A -90.000,B 90.000,C 0.000} C_DIS
LIN {X 47.377,Y -31.308,Z -44.636,A -90.000,B 90.000,C 0.000} C_DIS
LIN {X 47.817,Y -31.308,Z -44.653,A -90.000,B 90.000,C 0.000} C_DIS
LIN {X 48.448,Y -31.308,Z -44.716,A -90.000,B 90.000,C 0.000} C_DIS
LIN {X 49.145,Y -31.308,Z -44.821,A -90.000,B 90.000,C 0.000} C_DIS
LIN {X 49.591,Y -31.308,Z -44.911,A -90.000,B 90.000,C 0.000} C_DIS
LIN {X 50.739,Y -31.308,Z -45.185,A -90.000,B 90.000,C 0.000} C_DIS
LIN {X 51.173,Y -31.308,Z -45.323,A -90.000,B 90.000,C 0.000} C_DIS
LIN {X 51.615,Y -31.308,Z -45.476,A -90.000,B 90.000,C 0.000} C_DIS
LIN {X 52.147,Y -31.308,Z -45.700,A -90.000,B 90.000,C 0.000} C_DIS
LIN {X 52.563,Y -31.308,Z -45.885,A -90.000,B 90.000,C 0.000} C_DIS
LIN {X 53.026,Y -31.308,Z -46.096,A -90.000,B 90.000,C 0.000} C_DIS
LIN {X 53.447,Y -31.308,Z -46.299,A -90.000,B 90.000,C 0.000} C_DIS
LIN {X 54.096,Y -31.308,Z -46.630,A -90.000,B 90.000,C 0.000} C_DIS
LIN {X 54.564,Y -31.308,Z -46.886,A -90.000,B 90.000,C 0.000} C_DIS
LIN {X 54.961,Y -31.308,Z -47.132,A -90.000,B 90.000,C 0.000} C_DIS
LIN {X 55.960,Y -31.308,Z -47.865,A -90.000,B 90.000,C 0.000} C_DIS
LIN {X 57.479,Y -31.308,Z -48.968,A -90.000,B 90.000,C 0.000} C_DIS
LIN {X 57.847,Y -31.308,Z -49.255,A -90.000,B 90.000,C 0.000} C_DIS
LIN {X 59.463,Y -31.308,Z -50.671,A -90.000,B 90.000,C 0.000} C_DIS
LIN {X 60.135,Y -31.308,Z -51.255,A -90.000,B 90.000,C 0.000} C_DIS
LIN {X 61.772,Y -31.308,Z -52.799,A -90.000,B 90.000,C 0.000} C_DIS
LIN {X 62.291,Y -31.308,Z -53.284,A -90.000,B 90.000,C 0.000} C_DIS
LIN {X 63.750,Y -31.308,Z -54.631,A -90.000,B 90.000,C 0.000} C_DIS
LIN {X 64.419,Y -31.308,Z -55.254,A -90.000,B 90.000,C 0.000} C_DIS
LIN {X 65.570,Y -31.308,Z -56.228,A -90.000,B 90.000,C 0.000} C_DIS
LIN {X 66.782,Y -31.308,Z -57.226,A -90.000,B 90.000,C 0.000} C_DIS
LIN {X 68.502,Y -31.308,Z -58.635,A -90.000,B 90.000,C 0.000} C_DIS
LIN {X 68.585,Y -31.308,Z -58.701,A -90.000,B 90.000,C 0.000} C_DIS
LIN {X 69.703,Y -31.308,Z -59.651,A -90.000,B 90.000,C 0.000} C_DIS
LIN {X 70.761,Y -31.308,Z -60.617,A -90.000,B 90.000,C 0.000} C_DIS
LIN {X 71.053,Y -31.308,Z -60.908,A -90.000,B 90.000,C 0.000} C_DIS
LIN {X 72.379,Y -31.308,Z -62.326,A -90.000,B 90.000,C 0.000} C_DIS
LIN {X 72.676,Y -31.308,Z -62.653,A -90.000,B 90.000,C 0.000} C_DIS
LIN {X 73.127,Y -31.308,Z -63.222,A -90.000,B 90.000,C 0.000} C_DIS
LIN {X 73.890,Y -31.308,Z -64.162,A -90.000,B 90.000,C 0.000} C_DIS
LIN {X 74.030,Y -31.308,Z -64.347,A -90.000,B 90.000,C 0.000} C_DIS
LIN {X 74.249,Y -31.308,Z -64.650,A -90.000,B 90.000,C 0.000} C_DIS
LIN {X 74.791,Y -31.308,Z -65.459,A -90.000,B 90.000,C 0.000} C_DIS
LIN {X 74.951,Y -31.308,Z -65.702,A -90.000,B 90.000,C 0.000} C_DIS
LIN {X 75.115,Y -31.308,Z -65.918,A -90.000,B 90.000,C 0.000} C_DIS
LIN {X 75.372,Y -31.308,Z -66.276,A -90.000,B 90.000,C 0.000} C_DIS
LIN {X 75.605,Y -31.308,Z -66.647,A -90.000,B 90.000,C 0.000} C_DIS
LIN {X 76.069,Y -31.308,Z -67.272,A -90.000,B 90.000,C 0.000} C_DIS
LIN {X 76.348,Y -31.308,Z -67.660,A -90.000,B 90.000,C 0.000} C_DIS
LIN {X 76.812,Y -31.308,Z -68.343,A -90.000,B 90.000,C 0.000} C_DIS
LIN {X 77.027,Y -31.308,Z -68.605,A -90.000,B 90.000,C 0.000} C_DIS
LIN {X 77.171,Y -31.308,Z -68.797,A -90.000,B 90.000,C 0.000} C_DIS
LIN {X 77.290,Y -31.308,Z -68.966,A -90.000,B 90.000,C 0.000} C_DIS
LIN {X 77.618,Y -31.308,Z -69.369,A -90.000,B 90.000,C 0.000} C_DIS
LIN {X 78.386,Y -31.308,Z -70.345,A -90.000,B 90.000,C 0.000} C_DIS
LIN {X 78.570,Y -31.308,Z -70.580,A -90.000,B 90.000,C 0.000} C_DIS
LIN {X 78.792,Y -31.308,Z -69.914,A -90.000,B 90.000,C 0.000} C_DIS
LIN {X 79.195,Y -31.308,Z -68.754,A -90.000,B 90.000,C 0.000} C_DIS
LIN {X 79.783,Y -31.308,Z -67.276,A -90.000,B 90.000,C 0.000} C_DIS
LIN {X 80.450,Y -31.308,Z -65.762,A -90.000,B 90.000,C 0.000} C_DIS
LIN {X 80.650,Y -31.308,Z -65.325,A -90.000,B 90.000,C 0.000} C_DIS
LIN {X 81.438,Y -31.308,Z -63.804,A -90.000,B 90.000,C 0.000} C_DIS
LIN {X 81.456,Y -31.308,Z -63.773,A -90.000,B 90.000,C 0.000} C_DIS
LIN {X 81.684,Y -31.308,Z -63.383,A -90.000,B 90.000,C 0.000} C_DIS
LIN {X 82.705,Y -31.308,Z -61.742,A -90.000,B 90.000,C 0.000} C_DIS
LIN {X 84.243,Y -31.308,Z -59.630,A -90.000,B 90.000,C 0.000} C_DIS
LIN {X 85.740,Y -31.308,Z -57.848,A -90.000,B 90.000,C 0.000} C_DIS
LIN {X 86.059,Y -31.308,Z -57.494,A -90.000,B 90.000,C 0.000} C_DIS
LIN {X 87.795,Y -31.308,Z -55.685,A -90.000,B 90.000,C 0.000} C_DIS
LIN {X 87.886,Y -31.308,Z -55.601,A -90.000,B 90.000,C 0.000} C_DIS
LIN {X 87.890,Y -31.308,Z -55.246,A -90.000,B 90.000,C 0.000} C_DIS
LIN {X 87.910,Y -31.308,Z -55.019,A -90.000,B 90.000,C 0.000} C_DIS
LIN {X 88.111,Y -31.308,Z -53.973,A -90.000,B 90.000,C 0.000} C_DIS
LIN {X 88.203,Y -31.308,Z -52.661,A -90.000,B 90.000,C 0.000} C_DIS
LIN {X 88.264,Y -31.308,Z -52.386,A -90.000,B 90.000,C 0.000} C_DIS
LIN {X 88.401,Y -31.308,Z -51.844,A -90.000,B 90.000,C 0.000} C_DIS
LIN {X 88.435,Y -31.308,Z -51.681,A -90.000,B 90.000,C 0.000} C_DIS
LIN {X 88.506,Y -31.308,Z -51.400,A -90.000,B 90.000,C 0.000} C_DIS
LIN {X 88.813,Y -31.308,Z -50.529,A -90.000,B 90.000,C 0.000} C_DIS
LIN {X 88.940,Y -31.308,Z -50.201,A -90.000,B 90.000,C 0.000} C_DIS
LIN {X 89.212,Y -31.308,Z -49.603,A -90.000,B 90.000,C 0.000} C_DIS
LIN {X 89.503,Y -31.308,Z -48.988,A -90.000,B 90.000,C 0.000} C_DIS
LIN {X 89.983,Y -31.308,Z -48.040,A -90.000,B 90.000,C 0.000} C_DIS
LIN {X 90.379,Y -31.308,Z -47.346,A -90.000,B 90.000,C 0.000} C_DIS
LIN {X 90.570,Y -31.308,Z -47.023,A -90.000,B 90.000,C 0.000} C_DIS
LIN {X 90.797,Y -31.308,Z -46.690,A -90.000,B 90.000,C 0.000} C_DIS
LIN {X 91.451,Y -31.308,Z -45.745,A -90.000,B 90.000,C 0.000} C_DIS
LIN {X 91.776,Y -31.308,Z -45.327,A -90.000,B 90.000,C 0.000} C_DIS
LIN {X 92.140,Y -31.308,Z -44.884,A -90.000,B 90.000,C 0.000} C_DIS
LIN {X 92.425,Y -31.308,Z -44.548,A -90.000,B 90.000,C 0.000} C_DIS
LIN {X 93.141,Y -31.308,Z -43.760,A -90.000,B 90.000,C 0.000} C_DIS
LIN {X 93.573,Y -31.308,Z -43.323,A -90.000,B 90.000,C 0.000} C_DIS
LIN {X 94.147,Y -31.308,Z -42.781,A -90.000,B 90.000,C 0.000} C_DIS
LIN {X 94.495,Y -31.308,Z -42.469,A -90.000,B 90.000,C 0.000} C_DIS
LIN {X 95.044,Y -31.308,Z -41.996,A -90.000,B 90.000,C 0.000} C_DIS
LIN {X 95.335,Y -31.308,Z -41.758,A -90.000,B 90.000,C 0.000} C_DIS
LIN {X 95.539,Y -31.308,Z -41.594,A -90.000,B 90.000,C 0.000} C_DIS
LIN {X 96.530,Y -31.308,Z -40.872,A -90.000,B 90.000,C 0.000} C_DIS
LIN {X 96.931,Y -31.308,Z -40.606,A -90.000,B 90.000,C 0.000} C_DIS
LIN {X 97.490,Y -31.308,Z -40.262,A -90.000,B 90.000,C 0.000} C_DIS
LIN {X 97.909,Y -31.308,Z -40.014,A -90.000,B 90.000,C 0.000} C_DIS
LIN {X 98.835,Y -31.308,Z -39.510,A -90.000,B 90.000,C 0.000} C_DIS
LIN {X 100.266,Y -31.308,Z -38.830,A -90.000,B 90.000,C 0.000} C_DIS
LIN {X 102.092,Y -31.308,Z -38.003,A -90.000,B 90.000,C 0.000} C_DIS
LIN {X 103.303,Y -31.308,Z -37.461,A -90.000,B 90.000,C 0.000} C_DIS
LIN {X 104.492,Y -31.308,Z -36.936,A -90.000,B 90.000,C 0.000} C_DIS
LIN {X 105.385,Y -31.308,Z -36.559,A -90.000,B 90.000,C 0.000} C_DIS
LIN {X 106.897,Y -31.308,Z -35.959,A -90.000,B 90.000,C 0.000} C_DIS
LIN {X 107.419,Y -31.308,Z -35.761,A -90.000,B 90.000,C 0.000} C_DIS
LIN {X 107.891,Y -31.308,Z -35.592,A -90.000,B 90.000,C 0.000} C_DIS
LIN {X 108.328,Y -31.308,Z -35.445,A -90.000,B 90.000,C 0.000} C_DIS
LIN {X 108.757,Y -31.308,Z -35.330,A -90.000,B 90.000,C 0.000} C_DIS
LIN {X 109.231,Y -31.308,Z -35.224,A -90.000,B 90.000,C 0.000} C_DIS
LIN {X 109.677,Y -31.308,Z -35.165,A -90.000,B 90.000,C 0.000} C_DIS
LIN {X 110.108,Y -31.308,Z -35.113,A -90.000,B 90.000,C 0.000} C_DIS
LIN {X 110.605,Y -31.308,Z -35.105,A -90.000,B 90.000,C 0.000} C_DIS
LIN {X 110.949,Y -31.308,Z -35.117,A -90.000,B 90.000,C 0.000} C_DIS
LIN {X 111.439,Y -31.308,Z -35.159,A -90.000,B 90.000,C 0.000} C_DIS
LIN {X 112.077,Y -31.308,Z -35.279,A -90.000,B 90.000,C 0.000} C_DIS
LIN {X 112.419,Y -31.308,Z -35.366,A -90.000,B 90.000,C 0.000} C_DIS
LIN {X 112.894,Y -31.308,Z -35.509,A -90.000,B 90.000,C 0.000} C_DIS
LIN {X 113.055,Y -31.308,Z -35.560,A -90.000,B 90.000,C 0.000} C_DIS
LIN {X 113.520,Y -31.308,Z -35.753,A -90.000,B 90.000,C 0.000} C_DIS
LIN {X 113.993,Y -31.308,Z -35.980,A -90.000,B 90.000,C 0.000} C_DIS
LIN {X 114.426,Y -31.308,Z -36.215,A -90.000,B 90.000,C 0.000} C_DIS
LIN {X 114.554,Y -31.308,Z -36.295,A -90.000,B 90.000,C 0.000} C_DIS
LIN {X 114.958,Y -31.308,Z -36.571,A -90.000,B 90.000,C 0.000} C_DIS
LIN {X 115.089,Y -31.308,Z -36.677,A -90.000,B 90.000,C 0.000} C_DIS
LIN {X 115.435,Y -31.308,Z -36.969,A -90.000,B 90.000,C 0.000} C_DIS
LIN {X 115.525,Y -31.308,Z -37.051,A -90.000,B 90.000,C 0.000} C_DIS
LIN {X 115.852,Y -31.308,Z -37.389,A -90.000,B 90.000,C 0.000} C_DIS
LIN {X 116.084,Y -31.308,Z -37.637,A -90.000,B 90.000,C 0.000} C_DIS
LIN {X 116.439,Y -31.308,Z -38.088,A -90.000,B 90.000,C 0.000} C_DIS
LIN {X 116.700,Y -31.308,Z -38.500,A -90.000,B 90.000,C 0.000} C_DIS
LIN {X 116.922,Y -31.308,Z -38.948,A -90.000,B 90.000,C 0.000} C_DIS
LIN {X 117.061,Y -31.308,Z -39.255,A -90.000,B 90.000,C 0.000} C_DIS
LIN {X 117.114,Y -31.308,Z -39.392,A -90.000,B 90.000,C 0.000} C_DIS
LIN {X 117.260,Y -31.308,Z -39.781,A -90.000,B 90.000,C 0.000} C_DIS
LIN {X 117.387,Y -31.308,Z -40.266,A -90.000,B 90.000,C 0.000} C_DIS
LIN {X 117.462,Y -31.308,Z -40.593,A -90.000,B 90.000,C 0.000} C_DIS
LIN {X 117.544,Y -31.308,Z -41.135,A -90.000,B 90.000,C 0.000} C_DIS
LIN {X 117.594,Y -31.308,Z -41.508,A -90.000,B 90.000,C 0.000} C_DIS
LIN {X 117.631,Y -31.308,Z -41.891,A -90.000,B 90.000,C 0.000} C_DIS
LIN {X 117.657,Y -31.308,Z -42.408,A -90.000,B 90.000,C 0.000} C_DIS
LIN {X 117.668,Y -31.308,Z -42.707,A -90.000,B 90.000,C 0.000} C_DIS
LIN {X 117.663,Y -31.308,Z -42.890,A -90.000,B 90.000,C 0.000} C_DIS
LIN {X 117.651,Y -31.308,Z -43.202,A -90.000,B 90.000,C 0.000} C_DIS
LIN {X 117.605,Y -31.308,Z -43.748,A -90.000,B 90.000,C 0.000} C_DIS
LIN {X 117.564,Y -31.308,Z -44.134,A -90.000,B 90.000,C 0.000} C_DIS
LIN {X 117.486,Y -31.308,Z -44.651,A -90.000,B 90.000,C 0.000} C_DIS
LIN {X 117.394,Y -31.308,Z -45.135,A -90.000,B 90.000,C 0.000} C_DIS
LIN {X 117.256,Y -31.308,Z -45.754,A -90.000,B 90.000,C 0.000} C_DIS
LIN {X 117.114,Y -31.308,Z -46.230,A -90.000,B 90.000,C 0.000} C_DIS
LIN {X 116.900,Y -31.308,Z -46.938,A -90.000,B 90.000,C 0.000} C_DIS
LIN {X 116.538,Y -31.308,Z -47.877,A -90.000,B 90.000,C 0.000} C_DIS
LIN {X 116.372,Y -31.308,Z -48.278,A -90.000,B 90.000,C 0.000} C_DIS
LIN {X 115.857,Y -31.308,Z -49.383,A -90.000,B 90.000,C 0.000} C_DIS
LIN {X 115.206,Y -31.308,Z -50.683,A -90.000,B 90.000,C 0.000} C_DIS
LIN {X 114.605,Y -31.308,Z -51.874,A -90.000,B 90.000,C 0.000} C_DIS
LIN {X 113.924,Y -31.308,Z -53.266,A -90.000,B 90.000,C 0.000} C_DIS
LIN {X 113.276,Y -31.308,Z -54.687,A -90.000,B 90.000,C 0.000} C_DIS
LIN {X 112.799,Y -31.308,Z -55.830,A -90.000,B 90.000,C 0.000} C_DIS
LIN {X 112.741,Y -31.308,Z -55.983,A -90.000,B 90.000,C 0.000} C_DIS
LIN {X 112.213,Y -31.308,Z -57.388,A -90.000,B 90.000,C 0.000} C_DIS
LIN {X 111.674,Y -31.308,Z -59.009,A -90.000,B 90.000,C 0.000} C_DIS
LIN {X 111.250,Y -31.308,Z -60.481,A -90.000,B 90.000,C 0.000} C_DIS
LIN {X 110.694,Y -31.308,Z -62.515,A -90.000,B 90.000,C 0.000} C_DIS
LIN {X 110.152,Y -31.308,Z -64.440,A -90.000,B 90.000,C 0.000} C_DIS
LIN {X 110.012,Y -31.308,Z -64.909,A -90.000,B 90.000,C 0.000} C_DIS
LIN {X 109.336,Y -31.308,Z -67.075,A -90.000,B 90.000,C 0.000} C_DIS
LIN {X 108.512,Y -31.308,Z -69.376,A -90.000,B 90.000,C 0.000} C_DIS
LIN {X 107.585,Y -31.308,Z -71.708,A -90.000,B 90.000,C 0.000} C_DIS
LIN {X 107.383,Y -31.308,Z -72.197,A -90.000,B 90.000,C 0.000} C_DIS
LIN {X 106.407,Y -31.308,Z -74.435,A -90.000,B 90.000,C 0.000} C_DIS
LIN {X 105.792,Y -31.308,Z -75.720,A -90.000,B 90.000,C 0.000} C_DIS
LIN {X 105.388,Y -31.308,Z -76.556,A -90.000,B 90.000,C 0.000} C_DIS
LIN {X 104.136,Y -31.308,Z -78.889,A -90.000,B 90.000,C 0.000} C_DIS
LIN {X 103.962,Y -31.308,Z -79.191,A -90.000,B 90.000,C 0.000} C_DIS
LIN {X 103.041,Y -31.308,Z -80.752,A -90.000,B 90.000,C 0.000} C_DIS
LIN {X 102.188,Y -31.308,Z -82.093,A -90.000,B 90.000,C 0.000} C_DIS
LIN {X 100.190,Y -31.308,Z -85.085,A -90.000,B 90.000,C 0.000} C_DIS
LIN {X 99.004,Y -31.308,Z -86.839,A -90.000,B 90.000,C 0.000} C_DIS
LIN {X 98.934,Y -31.308,Z -87.198,A -90.000,B 90.000,C 0.000} C_DIS
LIN {X 98.870,Y -31.308,Z -87.909,A -90.000,B 90.000,C 0.000} C_DIS
LIN {X 98.812,Y -31.308,Z -88.402,A -90.000,B 90.000,C 0.000} C_DIS
LIN {X 98.692,Y -31.308,Z -90.326,A -90.000,B 90.000,C 0.000} C_DIS
LIN {X 98.676,Y -31.308,Z -90.730,A -90.000,B 90.000,C 0.000} C_DIS
LIN {X 98.648,Y -31.308,Z -91.471,A -90.000,B 90.000,C 0.000} C_DIS
LIN {X 98.563,Y -31.308,Z -92.796,A -90.000,B 90.000,C 0.000} C_DIS
LIN {X 98.493,Y -31.308,Z -93.822,A -90.000,B 90.000,C 0.000} C_DIS
LIN {X 98.465,Y -31.308,Z -94.087,A -90.000,B 90.000,C 0.000} C_DIS
LIN {X 98.398,Y -31.308,Z -94.642,A -90.000,B 90.000,C 0.000} C_DIS
LIN {X 98.337,Y -31.308,Z -95.105,A -90.000,B 90.000,C 0.000} C_DIS
LIN {X 98.266,Y -31.308,Z -95.533,A -90.000,B 90.000,C 0.000} C_DIS
LIN {X 98.152,Y -31.308,Z -96.005,A -90.000,B 90.000,C 0.000} C_DIS
LIN {X 97.983,Y -31.308,Z -96.653,A -90.000,B 90.000,C 0.000} C_DIS
LIN {X 97.905,Y -31.308,Z -96.977,A -90.000,B 90.000,C 0.000} C_DIS
LIN {X 97.800,Y -31.308,Z -97.337,A -90.000,B 90.000,C 0.000} C_DIS
LIN {X 97.766,Y -31.308,Z -97.442,A -90.000,B 90.000,C 0.000} C_DIS
LIN {X 97.688,Y -31.308,Z -97.715,A -90.000,B 90.000,C 0.000} C_DIS
LIN {X 97.573,Y -31.308,Z -98.098,A -90.000,B 90.000,C 0.000} C_DIS
LIN {X 97.530,Y -31.308,Z -98.264,A -90.000,B 90.000,C 0.000} C_DIS
LIN {X 97.292,Y -31.308,Z -98.984,A -90.000,B 90.000,C 0.000} C_DIS
LIN {X 97.255,Y -31.308,Z -99.106,A -90.000,B 90.000,C 0.000} C_DIS
LIN {X 96.937,Y -31.308,Z -100.391,A -90.000,B 90.000,C 0.000} C_DIS
LIN {X 96.738,Y -31.308,Z -101.325,A -90.000,B 90.000,C 0.000} C_DIS
LIN {X 96.640,Y -31.308,Z -101.804,A -90.000,B 90.000,C 0.000} C_DIS
LIN {X 96.411,Y -31.308,Z -103.133,A -90.000,B 90.000,C 0.000} C_DIS
LIN {X 96.381,Y -31.308,Z -103.286,A -90.000,B 90.000,C 0.000} C_DIS
LIN {X 96.227,Y -31.308,Z -104.440,A -90.000,B 90.000,C 0.000} C_DIS
LIN {X 96.213,Y -31.308,Z -105.098,A -90.000,B 90.000,C 0.000} C_DIS
LIN {X 96.242,Y -31.308,Z -105.373,A -90.000,B 90.000,C 0.000} C_DIS
LIN {X 96.291,Y -31.308,Z -105.893,A -90.000,B 90.000,C 0.000} C_DIS
LIN {X 96.379,Y -31.308,Z -106.422,A -90.000,B 90.000,C 0.000} C_DIS
LIN {X 96.461,Y -31.308,Z -106.961,A -90.000,B 90.000,C 0.000} C_DIS
LIN {X 96.627,Y -31.308,Z -108.191,A -90.000,B 90.000,C 0.000} C_DIS
LIN {X 96.694,Y -31.308,Z -109.268,A -90.000,B 90.000,C 0.000} C_DIS
LIN {X 96.725,Y -31.308,Z -109.720,A -90.000,B 90.000,C 0.000} C_DIS
LIN {X 96.750,Y -31.308,Z -110.160,A -90.000,B 90.000,C 0.000} C_DIS
LIN {X 96.788,Y -31.308,Z -111.586,A -90.000,B 90.000,C 0.000} C_DIS
LIN {X 96.801,Y -31.308,Z -111.939,A -90.000,B 90.000,C 0.000} C_DIS
LIN {X 96.824,Y -31.308,Z -113.710,A -90.000,B 90.000,C 0.000} C_DIS
LIN {X 96.828,Y -31.308,Z -113.913,A -90.000,B 90.000,C 0.000} C_DIS
LIN {X 96.859,Y -31.308,Z -116.045,A -90.000,B 90.000,C 0.000} C_DIS
LIN {X 96.866,Y -31.308,Z -116.306,A -90.000,B 90.000,C 0.000} C_DIS
LIN {X 96.906,Y -31.308,Z -118.212,A -90.000,B 90.000,C 0.000} C_DIS
LIN {X 96.960,Y -31.308,Z -120.436,A -90.000,B 90.000,C 0.000} C_DIS
LIN {X 96.997,Y -31.308,Z -122.660,A -90.000,B 90.000,C 0.000} C_DIS
LIN {X 96.990,Y -31.308,Z -124.906,A -90.000,B 90.000,C 0.000} C_DIS
LIN {X 96.987,Y -31.308,Z -125.037,A -90.000,B 90.000,C 0.000} C_DIS
LIN {X 96.912,Y -31.308,Z -127.170,A -90.000,B 90.000,C 0.000} C_DIS
LIN {X 96.857,Y -31.308,Z -128.038,A -90.000,B 90.000,C 0.000} C_DIS
LIN {X 96.778,Y -31.308,Z -129.370,A -90.000,B 90.000,C 0.000} C_DIS
LIN {X 96.687,Y -31.308,Z -130.518,A -90.000,B 90.000,C 0.000} C_DIS
LIN {X 96.593,Y -31.308,Z -131.763,A -90.000,B 90.000,C 0.000} C_DIS
LIN {X 96.469,Y -31.308,Z -133.256,A -90.000,B 90.000,C 0.000} C_DIS
LIN {X 96.371,Y -31.308,Z -134.482,A -90.000,B 90.000,C 0.000} C_DIS
LIN {X 96.219,Y -31.308,Z -136.426,A -90.000,B 90.000,C 0.000} C_DIS
LIN {X 96.121,Y -31.308,Z -137.658,A -90.000,B 90.000,C 0.000} C_DIS
LIN {X 95.947,Y -31.308,Z -139.755,A -90.000,B 90.000,C 0.000} C_DIS
LIN {X 95.797,Y -31.308,Z -141.520,A -90.000,B 90.000,C 0.000} C_DIS
LIN {X 95.579,Y -31.308,Z -143.786,A -90.000,B 90.000,C 0.000} C_DIS
LIN {X 95.440,Y -31.308,Z -145.198,A -90.000,B 90.000,C 0.000} C_DIS
LIN {X 95.168,Y -31.308,Z -147.519,A -90.000,B 90.000,C 0.000} C_DIS
LIN {X 95.000,Y -31.308,Z -148.922,A -90.000,B 90.000,C 0.000} C_DIS
LIN {X 94.663,Y -31.308,Z -151.206,A -90.000,B 90.000,C 0.000} C_DIS
LIN {X 94.457,Y -31.308,Z -152.557,A -90.000,B 90.000,C 0.000} C_DIS
LIN {X 94.057,Y -31.308,Z -154.809,A -90.000,B 90.000,C 0.000} C_DIS
LIN {X 93.811,Y -31.308,Z -156.142,A -90.000,B 90.000,C 0.000} C_DIS
LIN {X 93.264,Y -31.308,Z -158.780,A -90.000,B 90.000,C 0.000} C_DIS
LIN {X 92.974,Y -31.308,Z -160.128,A -90.000,B 90.000,C 0.000} C_DIS
LIN {X 92.457,Y -31.308,Z -162.327,A -90.000,B 90.000,C 0.000} C_DIS
LIN {X 92.115,Y -31.308,Z -163.724,A -90.000,B 90.000,C 0.000} C_DIS
LIN {X 91.551,Y -31.308,Z -165.900,A -90.000,B 90.000,C 0.000} C_DIS
LIN {X 91.148,Y -31.308,Z -167.380,A -90.000,B 90.000,C 0.000} C_DIS
LIN {X 90.569,Y -31.308,Z -169.463,A -90.000,B 90.000,C 0.000} C_DIS
LIN {X 89.550,Y -31.308,Z -172.953,A -90.000,B 90.000,C 0.000} C_DIS
LIN {X 89.074,Y -31.308,Z -174.504,A -90.000,B 90.000,C 0.000} C_DIS
LIN {X 88.510,Y -31.308,Z -176.385,A -90.000,B 90.000,C 0.000} C_DIS
LIN {X 88.018,Y -31.308,Z -177.950,A -90.000,B 90.000,C 0.000} C_DIS
LIN {X 87.781,Y -31.308,Z -178.699,A -90.000,B 90.000,C 0.000} C_DIS
LIN {X 87.106,Y -31.308,Z -180.933,A -90.000,B 90.000,C 0.000} C_DIS
LIN {X 86.923,Y -31.308,Z -181.506,A -90.000,B 90.000,C 0.000} C_DIS
LIN {X 86.267,Y -31.308,Z -183.678,A -90.000,B 90.000,C 0.000} C_DIS
LIN {X 86.128,Y -31.308,Z -184.113,A -90.000,B 90.000,C 0.000} C_DIS
LIN {X 85.486,Y -31.308,Z -186.256,A -90.000,B 90.000,C 0.000} C_DIS
LIN {X 85.392,Y -31.308,Z -186.553,A -90.000,B 90.000,C 0.000} C_DIS
LIN {X 84.978,Y -31.308,Z -187.963,A -90.000,B 90.000,C 0.000} C_DIS
LIN {X 84.884,Y -31.308,Z -188.349,A -90.000,B 90.000,C 0.000} C_DIS
LIN {X 84.767,Y -31.308,Z -188.855,A -90.000,B 90.000,C 0.000} C_DIS
LIN {X 84.229,Y -31.308,Z -190.814,A -90.000,B 90.000,C 0.000} C_DIS
LIN {X 84.045,Y -31.308,Z -191.612,A -90.000,B 90.000,C 0.000} C_DIS
LIN {X 83.828,Y -31.308,Z -192.484,A -90.000,B 90.000,C 0.000} C_DIS
LIN {X 83.527,Y -31.308,Z -193.575,A -90.000,B 90.000,C 0.000} C_DIS
LIN {X 83.028,Y -31.308,Z -195.641,A -90.000,B 90.000,C 0.000} C_DIS
LIN {X 82.767,Y -31.308,Z -196.555,A -90.000,B 90.000,C 0.000} C_DIS
LIN {X 82.090,Y -31.308,Z -199.165,A -90.000,B 90.000,C 0.000} C_DIS
LIN {X 82.048,Y -31.308,Z -199.344,A -90.000,B 90.000,C 0.000} C_DIS
LIN {X 81.991,Y -31.308,Z -199.591,A -90.000,B 90.000,C 0.000} C_DIS
LIN {X 81.879,Y -31.308,Z -200.121,A -90.000,B 90.000,C 0.000} C_DIS
LIN {X 81.588,Y -31.308,Z -201.427,A -90.000,B 90.000,C 0.000} C_DIS
LIN {X 81.022,Y -31.308,Z -203.687,A -90.000,B 90.000,C 0.000} C_DIS
LIN {X 80.243,Y -31.308,Z -207.167,A -90.000,B 90.000,C 0.000} C_DIS
LIN {X 79.967,Y -31.308,Z -208.215,A -90.000,B 90.000,C 0.000} C_DIS
LIN {X 79.308,Y -31.308,Z -211.086,A -90.000,B 90.000,C 0.000} C_DIS
LIN {X 78.870,Y -31.308,Z -213.140,A -90.000,B 90.000,C 0.000} C_DIS
LIN {X 78.655,Y -31.308,Z -214.302,A -90.000,B 90.000,C 0.000} C_DIS
LIN {X 78.348,Y -31.308,Z -215.923,A -90.000,B 90.000,C 0.000} C_DIS
LIN {X 77.865,Y -31.308,Z -218.171,A -90.000,B 90.000,C 0.000} C_DIS
LIN {X 77.606,Y -31.308,Z -219.287,A -90.000,B 90.000,C 0.000} C_DIS
LIN {X 77.228,Y -31.308,Z -221.769,A -90.000,B 90.000,C 0.000} C_DIS
LIN {X 76.875,Y -31.308,Z -223.594,A -90.000,B 90.000,C 0.000} C_DIS
LIN {X 76.599,Y -31.308,Z -224.863,A -90.000,B 90.000,C 0.000} C_DIS
LIN {X 75.786,Y -31.308,Z -228.183,A -90.000,B 90.000,C 0.000} C_DIS
LIN {X 75.591,Y -31.308,Z -229.137,A -90.000,B 90.000,C 0.000} C_DIS
LIN {X 74.638,Y -31.308,Z -232.610,A -90.000,B 90.000,C 0.000} C_DIS
LIN {X 74.106,Y -31.308,Z -234.841,A -90.000,B 90.000,C 0.000} C_DIS
LIN {X 73.342,Y -31.308,Z -237.248,A -90.000,B 90.000,C 0.000} C_DIS
LIN {X 72.290,Y -31.308,Z -240.823,A -90.000,B 90.000,C 0.000} C_DIS
LIN {X 72.195,Y -31.308,Z -241.088,A -90.000,B 90.000,C 0.000} C_DIS
LIN {X 71.678,Y -31.308,Z -242.472,A -90.000,B 90.000,C 0.000} C_DIS
LIN {X 71.277,Y -31.308,Z -243.561,A -90.000,B 90.000,C 0.000} C_DIS
LIN {X 71.277,Y -60.000,Z -243.561,A -90.000,B 90.000,C 0.000} C_DIS
